(* IEC 61131-3 sources: elnaProjects/ElpcLogic/PomarKc7Changed/build_USO_ecl/_ (part 7) *)

  (* [A2-15, AI1-3]  TOpornoYpornogoPodshipnikaEDT_2 *)
  stAI_Ini(data_Ini := TRUE,  dLL := 0.0, dHL := 100.0,
  ISVALIDREF_HA := TRUE, ISVALIDREF_HW := TRUE, dHA := 80.0, dHW := 75.0, aperturFilter:= 0.5, dMaxChangeSpeed := 10.0,
  strAI := ai.Toy_podshipnika_EDT_2);
  inits := inits + BOOL_TO_UINT(stAI_Ini.Init);

  (********************************************* Модуль A3-1 ******************************************************)

  (* [A3-1, AI2-0]  TOpornoYpornogoPodshipnikaKolesaRedEDT_3 *)
  stAI_Ini(data_Ini := TRUE,  dLL := 0.0, dHL := 100.0,
  ISVALIDREF_HA := TRUE, ISVALIDREF_HW := TRUE, dHA := 80.0, dHW := 75.0, aperturFilter:= 0.5, dMaxChangeSpeed := 10.0,
  strAI := ai.Toy_podshipnika_kol_EDT_3);
  inits := inits + BOOL_TO_UINT(stAI_Ini.Init);

  (* [A3-1, AI2-1] TOpornoYpornogoPodshipnikaKolesaRedHT_4 *)
  stAI_Ini(data_Ini := TRUE,  dLL := 0.0, dHL := 100.0,
  ISVALIDREF_HA := TRUE, ISVALIDREF_HW := TRUE, dHA := 80.0, dHW := 75.0, aperturFilter:= 0.5, dMaxChangeSpeed := 10.0,
  strAI := ai.Toy_podshipnika_kol_EDT_4);
  inits := inits + BOOL_TO_UINT(stAI_Ini.Init);

  (* [A3-1, AI2-2] TOpornogoPodshipnikaShesterniReduktoraT_5 *)
  stAI_Ini(data_Ini := TRUE,  dLL := 0.0, dHL := 100.0,
  ISVALIDREF_HA := TRUE, ISVALIDREF_HW := TRUE, dHA := 80.0, dHW := 75.0, aperturFilter:= 0.5, dMaxChangeSpeed := 10.0,
  strAI := ai.Toy_podshipnika_shest_red_EDT_5);
  inits := inits + BOOL_TO_UINT(stAI_Ini.Init);

  (* [A3-1, AI2-3] TOpornogoPodshipnikaReduktoraHT_6 *)
  stAI_Ini(data_Ini := TRUE,  dLL := 0.0, dHL := 100.0,
  ISVALIDREF_HA := TRUE, ISVALIDREF_HW := TRUE, dHA := 80.0, dHW := 75.0, aperturFilter:= 0.5, dMaxChangeSpeed := 10.0,
  strAI := ai.Ty_podshipnika_red_EDT_6);
  inits := inits + BOOL_TO_UINT(stAI_Ini.Init);

  (********************************************* Модуль A3-2 ******************************************************)

  (* [A3-2, AI3-01]  TOpornoYpornogoPodshipnikaNagnetateljaT_7_1 *)
  stAI_Ini(data_Ini := TRUE,  dLL := 0.0, dHL := 100.0,
  ISVALIDREF_HA := TRUE, ISVALIDREF_HW := TRUE, dHA := 80.0, dHW := 75.0, aperturFilter:= 0.5, dMaxChangeSpeed := 10.0,
  strAI := ai.Ty_podshipnika_nagnet_EDT_7_1);
  inits := inits + BOOL_TO_UINT(stAI_Ini.Init);

  (* [A3-2, AI3-01]  TOpornoYpornogoPodshipnikaNagnetateljaT_7_2 *)
  stAI_Ini(data_Ini := TRUE,  dLL := 0.0, dHL := 100.0,
  ISVALIDREF_HA := TRUE, ISVALIDREF_HW := TRUE, dHA := 80.0, dHW := 75.0, aperturFilter:= 0.5, dMaxChangeSpeed := 10.0,
  strAI := ai.Ty_podshipnika_nagnet_EDT_7_2);
  inits := inits + BOOL_TO_UINT(stAI_Ini.Init);

  (* [A3-2, AI3-2]  TOpornoYpornogoPodshipnikaSvobodnogoKoncaNT_8_1 *)
  stAI_Ini(data_Ini := TRUE,  dLL := 0.0, dHL := 100.0,
  ISVALIDREF_HA := TRUE, ISVALIDREF_HW := TRUE, dHA := 80.0, dHW := 75.0, aperturFilter:= 0.5, dMaxChangeSpeed := 10.0,
  strAI := ai.Toy_podshipnika_svobod_konca_EDT_8_1);
  inits := inits + BOOL_TO_UINT(stAI_Ini.Init);

  (* [A3-2, AI3-2]  TOpornoYpornogoPodshipnikaSvobodnogoKoncaNT_8_2 *)
  stAI_Ini(data_Ini := TRUE,  dLL := 0.0, dHL := 100.0,
  ISVALIDREF_HA := TRUE, ISVALIDREF_HW := TRUE, dHA := 80.0, dHW := 75.0, aperturFilter:= 0.5, dMaxChangeSpeed := 10.0,
  strAI := ai.Toy_podshipnika_svobod_konca_EDT_8_2);
  inits := inits + BOOL_TO_UINT(stAI_Ini.Init);

  (********************************************* Модуль A3-3 ******************************************************)

  (* [A3-3, AI4-1]  TYpornogoPodshipnikaRavKolodokHT_9_1 *)
  stAI_Ini(data_Ini := TRUE,  dLL := 0.0, dHL := 100.0,
  ISVALIDREF_HA := TRUE, ISVALIDREF_HW := TRUE, dHA := 80.0, dHW := 75.0, aperturFilter:= 0.5, dMaxChangeSpeed := 10.0,
  strAI := ai.Toy_podshipnika_rab_kol_EDT_9_1);
  inits := inits + BOOL_TO_UINT(stAI_Ini.Init);

  (* [A3-3, AI4-1]  TYpornogoPodshipnikaRavKolodokHT_9_2 *)
  stAI_Ini(data_Ini := TRUE,  dLL := 0.0, dHL := 100.0,
  ISVALIDREF_HA := TRUE, ISVALIDREF_HW := TRUE, dHA := 80.0, dHW := 75.0, aperturFilter:= 0.5, dMaxChangeSpeed := 10.0,
  strAI := ai.Toy_podshipnika_rab_kol_EDT_9_2);
  inits := inits + BOOL_TO_UINT(stAI_Ini.Init);

  (* [A3-3, AI4-3] TYpornogoPodshipnikaNerabKolodokHT_10_1 *)
  stAI_Ini(data_Ini := TRUE,  dLL := 0.0, dHL := 100.0,
  ISVALIDREF_HA := TRUE, ISVALIDREF_HW := TRUE, dHA := 80.0, dHW := 75.0, aperturFilter:= 0.5, dMaxChangeSpeed := 10.0,
  strAI := ai.Toy_podshipnika_nerab_kol_EDT_10_1);
  inits := inits + BOOL_TO_UINT(stAI_Ini.Init);

  (* [A3-3, AI4-3] TYpornogoPodshipnikaNerabKolodokHT_10_2 *)
  stAI_Ini(data_Ini := TRUE,  dLL := 0.0, dHL := 100.0,
  ISVALIDREF_HA := TRUE, ISVALIDREF_HW := TRUE, dHA := 80.0, dHW := 75.0, aperturFilter:= 0.5, dMaxChangeSpeed := 10.0,
  strAI := ai.Toy_podshipnika_nerab_kol_EDT_10_2);
  inits := inits + BOOL_TO_UINT(stAI_Ini.Init);

  (********************************************* Модуль A3-4 ******************************************************)
  (* [A3-4, AI5-0] THolodnogoVozduhaEDKanall *)
  stAI_Ini(data_Ini := TRUE,  dLL := 0.0, dHL := 100.0,
  ISVALIDREF_HW := TRUE, dHW := 60.0, aperturFilter:= 0.5,
  strAI := ai.Tholodnogo_vozduha_ED_kanal_1);
  inits := inits + BOOL_TO_UINT(stAI_Ini.Init);

  (* [A3-4, AI5-1] THolodnogoVozduhaEDKanal2 *)
  stAI_Ini(data_Ini := TRUE,  dLL := 0.0, dHL := 100.0,
  ISVALIDREF_HW := TRUE, dHW := 60.0, aperturFilter:= 0.5,
  strAI := ai.Tholodnogo_vozduha_ED_kanal_2);
  inits := inits + BOOL_TO_UINT(stAI_Ini.Init);

  (* [A3-4, AI5-2]  TGorjachegoVozduhaEDKanall *)
  stAI_Ini(data_Ini := TRUE,  dLL := 0.0, dHL := 100.0,
  ISVALIDREF_HW := TRUE, dHW := 70.0, aperturFilter:= 0.5,
  strAI := ai.Tgorjachego_vozduha_ED_kanal_1);
  inits := inits + BOOL_TO_UINT(stAI_Ini.Init);

  (* [A3-4, AI5-3] TGorjachegoVozduhaEDKanal2 *)
  stAI_Ini(data_Ini := TRUE,  dLL := 0.0, dHL := 100.0,
  ISVALIDREF_HW := TRUE, dHW := 70.0, aperturFilter:= 0.5,
  strAI := ai.Tgorjachego_vozduha_ED_kanal_2);
  inits := inits + BOOL_TO_UINT(stAI_Ini.Init);

  (********************************************* Модуль A3-5 ******************************************************)

  (* [A3-5, AI6-0] TNArujnogoVozduha *)
  stAI_Ini(data_Ini := TRUE,  dLL := -50.0, dHL := 100.0,
  ISVALIDREF_HW := TRUE, dHW := 70.0, aperturFilter:= 0.5,
  strAI := ai.Tnarujnogo_vozduha);
  inits := inits + BOOL_TO_UINT(stAI_Ini.Init);

  (* [A3-5, AI6-1]  TgazaNaVhodeH *)
  stAI_Ini(data_Ini := TRUE,  dLL := -50.0, dHL := 100.0,
  ISVALIDREF_HW := TRUE, dHW := 80.0, aperturFilter:= 0.5,
  strAI := ai.Tgaza_na_vhode_H);
  inits := inits + BOOL_TO_UINT(stAI_Ini.Init);

  (* [A3-5, AI6-2] TgazaNaVyhodeH *)
  stAI_Ini(data_Ini := TRUE,  dLL := -50.0, dHL := 100.0,
  ISVALIDREF_HW := TRUE, ISVALIDREF_HA := TRUE, dHa :=90.0, dHW := 80.0, aperturFilter:= 0.5, dMaxChangeSpeed := 10.0,
  strAI := ai.Tgaza_na_vyhode_H);
  inits := inits + BOOL_TO_UINT(stAI_Ini.Init);

  (********************************************* Модуль A3-6 ******************************************************)
  (* [A3-6, AI7-0] TMasladoAVOM *)
  stAI_Ini(data_Ini := TRUE,  dLL := 0.0, dHL := 150.0,
  ISVALIDREF_HW := TRUE, dHW := 55.0, aperturFilter:= 0.5,
  strAI := ai.Tmasla_do_AVOM);
  inits := inits + BOOL_TO_UINT(stAI_Ini.Init);

  (* [A3-6, AI7-1] TMaslaPosleAVOM *)
  stAI_Ini(data_Ini := TRUE,  dLL := 0.0, dHL := 150.0,
  ISVALIDREF_HW := TRUE, dHW := 55.0, aperturFilter:= 0.5, dMaxChangeSpeed := 10.0,
  strAI := ai.Tmasla_posle_AVOM);
  inits := inits + BOOL_TO_UINT(stAI_Ini.Init);
  (********************************************* Модуль A3-8 ******************************************************)
  (* [A3-8, AI9-0]  TMaslaMB *)
  stAI_Ini(data_Ini := TRUE,  dLL := 0.0, dHL := 150.0,
  ISVALIDREF_LW := TRUE, dLW := 25.0, aperturFilter:= 0.5, dMaxChangeSpeed := 10.0,
  strAI := ai.Tmasla_MB);
  inits := inits + BOOL_TO_UINT(stAI_Ini.Init);

  (* [A3-6, AI7-2] TMaslaMB_TEN *)
  stAI_Ini(data_Ini := TRUE,  dLL := 0.0, dHL := 100.0,
  ISVALIDREF_HW := TRUE, dHW := 50.0, aperturFilter:= 0.5, dMaxChangeSpeed := 10.0,
  strAI := ai.Tmasla_MB_TEN);
  inits := inits + BOOL_TO_UINT(stAI_Ini.Init);

  (* [A3-8, AI9-1]  TEmperatura_v_SHU *)
  stAI_Ini(data_Ini := TRUE,  dLL := -40.0, dHL := 100.0, CurrentShotCircuit := 20320.0, CurrentBreakCircuit := 3680.0,
  aperturFilter:= 0.5, strAI := ai.Tshu);
  inits := inits + BOOL_TO_UINT(stAI_Ini.Init);

  (* [A3-8, AI9-2]  DavlenijaMasloSmNizkoe *)
  stAI_Ini(data_Ini := TRUE,  dLL := 0.0, dHL := 250.0,
  ISVALIDREF_LW := TRUE, ISVALIDREF_LA := TRUE, dLW := 50.0, dLA := 25.0,  CurrentShotCircuit := 20240.0, CurrentBreakCircuit := 3760.0,  aperturFilter:= 0.5,
  strAI := ai.Pmaslo_sm_nizkoe);
  inits := inits + BOOL_TO_UINT(stAI_Ini.Init);

  (* [A3-8, AI9-3]  PerepadDavlenieNaMasloFiltre *)
  stAI_Ini(data_Ini := TRUE,  dLL := 0.0, dHL := 250.0,
  ISVALIDREF_HW := TRUE, dHW := 150.0, CurrentShotCircuit := 20240.0, CurrentBreakCircuit := 3760.0, aperturFilter:= 0.5,
  strAI := ai.dPgaza_na_maslo_filtre);
  inits := inits + BOOL_TO_UINT(stAI_Ini.Init);

  (********************************************* Модуль A3-9 ******************************************************)
  (* [A3-9, AI10-0]  DavlenijaMasloSmVysokoe *)
  stAI_Ini(data_Ini := TRUE,  dLL := 0.0, dHL := 1000.0,
  ISVALIDREF_LW := TRUE, ISVALIDREF_LA := TRUE, dLW := 300.0, dLA := 250.0, CurrentShotCircuit := 20240.0, CurrentBreakCircuit := 3760.0, aperturFilter:= 0.5,
  strAI := ai.Pmaslo_sm_vysokoe);
  inits := inits + BOOL_TO_UINT(stAI_Ini.Init);

  (* [A3-9, AI10-1]  DavlenijaMaslaPosleGNS *)
  stAI_Ini(data_Ini := TRUE,  dLL := 0.0, dHL := 250.0, aperturFilter:= 0.5, CurrentShotCircuit := 20240.0, CurrentBreakCircuit := 3760.0,
  ISVALIDREF_LW := TRUE, ISVALIDREF_HW := TRUE,
  dLW := 187.0, dHW := 242.0,
  strAI := ai.Pmasla_posle_GNS);
  inits := inits + BOOL_TO_UINT(stAI_Ini.Init);

  (* [A3-9, AI10-2] DavlenijaMaslaPosleNU *)
  stAI_Ini(data_Ini := TRUE,  dLL := 0.0, dHL := 10.0, aperturFilter:= 0.5, CurrentShotCircuit := 20240.0, CurrentBreakCircuit := 3760.0,
  ISVALIDREF_LW := TRUE, dLW := 3.0,
  strAI := ai.Pmasla_posle_NU);
  inits := inits + BOOL_TO_UINT(stAI_Ini.Init);

  (********************************************* Модуль A3-10 ******************************************************)
  (* [A3-10, AI11-0] PerepadDavlenieNaKonfuzore *)
  stAI_Ini(data_Ini := TRUE,  dLL := 0.0, dHL := 250.0,
  ISVALIDREF_LW := TRUE, dLW := 15.0, aperturFilter:= 0.5, CurrentShotCircuit := 20240.0, CurrentBreakCircuit := 3760.0,
  strAI := ai.dPgaza_na_konfuzore);
  inits := inits + BOOL_TO_UINT(stAI_Ini.Init);

  (* [A3-10, AI11-1] OsSdvigNagnetatelja_Plus *)
  stAI_Ini(data_Ini := TRUE,  dLL := 0.0, dHL := 1000.0,
  ISVALIDREF_HA := TRUE, ISVALIDREF_HW := TRUE, dHW := 200.0, dHA := 300.0, aperturFilter := 0.5, CurrentShotCircuit := 20240.0, CurrentBreakCircuit := 3760.0,
  strAI := ai.Os_sdvig_nagnetatelja_plus);
  inits := inits + BOOL_TO_UINT(stAI_Ini.Init);

  (* [A3-10, AI11-2] OsSdvigNagnetatelja_Minus *)
  stAI_Ini(data_Ini := TRUE,  dLL := 0.0, dHL := 1600.0,
  ISVALIDREF_LW := TRUE, dLW := 150.0, ISVALIDREF_LA := TRUE, dLA := 100.0, aperturFilter := 0.5, CurrentShotCircuit := 20240.0, CurrentBreakCircuit := 3760.0,
  strAI := ai.Os_sdvig_nagnetatelja_minus);
  inits := inits + BOOL_TO_UINT(stAI_Ini.Init);

  (* [A3-10, AI11-3] PerepadDavlenieMasloGaz *)
  stAI_Ini(data_Ini := TRUE, dLL := 0.0, dHL := 1600.0,
  ISVALIDREF_LW := TRUE, ISVALIDREF_LA := TRUE, dLW := 150.0, dLa := 100.0, aperturFilter:= 0.5, CurrentShotCircuit := 20240.0, CurrentBreakCircuit := 3760.0,
  strAI := ai.dPmaslo_gaz);
  inits := inits + BOOL_TO_UINT(stAI_Ini.Init);

  (********************************************* Модуль A3-11 ******************************************************)
  (* [A3-11, AI12-0]  DGazaNaVhodeNagnetatelja *)
  stAI_Ini(data_Ini := TRUE,  dLL := 0.0, dHL := 10.0,
  ISVALIDREF_LW := TRUE, dLW := 4.895, aperturFilter := 0.5, CurrentShotCircuit := 20240.0, CurrentBreakCircuit := 3760.0,
  strAI := ai.Pgaza_na_vhode_nagnetatelia);
  inits := inits + BOOL_TO_UINT(stAI_Ini.Init);

  (* [A3-11, AI12-1]  DGazaNaVyhodeNagnetatelja *)
  stAI_Ini(data_Ini := TRUE,  dLL := 0.0, dHL := 10.0,
  ISVALIDREF_HA := TRUE, ISVALIDREF_HW := TRUE, dLA := 7.653, dHW := 7.55, aperturFilter := 0.5, CurrentShotCircuit := 20240.0, CurrentBreakCircuit := 3760.0,
  strAI := ai.Pgaza_na_vyhode_nagnetatelia);
  inits := inits + BOOL_TO_UINT(stAI_Ini.Init);

  (* [A3-11, AI12-3]  DavlenieImpulsGaz *)
  stAI_Ini(data_Ini := TRUE,  dLL := 0.0, dHL := 10.0,
  ISVALIDREF_LW := TRUE, dLW := 5.0, aperturFilter := 0.5, CurrentShotCircuit := 20240.0, CurrentBreakCircuit := 3760.0,
  strAI := ai.Pimpuls_gaz);
  inits := inits + BOOL_TO_UINT(stAI_Ini.Init);

  (********************************************* Модуль A3-12 ******************************************************)
  (* [A3-12, AI13-0] YrovenMaslaMB *)
  stAI_Ini(data_Ini := TRUE,  dLL := 190.0, dHL := 885.0,
  ISVALIDREF_LW := TRUE, dLW := 530.0, aperturFilter := 0.5,  CurrentShotCircuit := 20240.0, CurrentBreakCircuit := 3760.0,
  strAI := ai.Yroven_masla_MB);
  inits := inits + BOOL_TO_UINT(stAI_Ini.Init);

  (********************************************* Модуль A3-13 ******************************************************)
  (* [A3-13, AI14-0]  Kontrol_per220V *)
  stAI_Ini(data_Ini := TRUE,  dLL := 0.0, dHL := 250.0,
  ISVALIDREF_LW := TRUE, ISVALIDREF_HW := TRUE, dLW := 187.0, dHW := 242.0, aperturFilter := 0.5, CurrentShotCircuit := 20240.0, CurrentBreakCircuit := 3760.0,
  strAI := ai.Kontrol_per_220V);
  inits := inits + BOOL_TO_UINT(stAI_Ini.Init);

  (* [A3-13, AI14-1]  Kontrol_post220V *)
  stAI_Ini(data_Ini := TRUE,  dLL := 0.0, dHL := 250.0,
  ISVALIDREF_HW := TRUE, ISVALIDREF_LW := TRUE, dHW := 242.0, dLW := 187.0, aperturFilter := 0.5, CurrentShotCircuit := 20240.0, CurrentBreakCircuit := 3760.0,
  strAI := ai.Kontrol_post_220V);
  inits := inits + BOOL_TO_UINT(stAI_Ini.Init);

  (* [A3-13, AI14-2]  VibroSkorostOPED_T1 *)
  stAI_Ini(data_Ini := TRUE,  dLL := 0.0, dHL := 25.0,
  ISVALIDREF_HW := TRUE, ISVALIDREF_HA := TRUE, dHW := 11.0, dHA := 18.0, aperturFilter := 0.5, CurrentShotCircuit := 20240.0, CurrentBreakCircuit := 3760.0,
  strAI := ai.Vibro_skorost_OPED_T1);
  inits := inits + BOOL_TO_UINT(stAI_Ini.Init);

  (* [A3-13, AI14-3]  VibroSkorostOYPED_T2 *)
  stAI_Ini(data_Ini := TRUE,  dLL := 0.0, dHL := 25.0,
  ISVALIDREF_HW := TRUE, ISVALIDREF_HA := TRUE, dHW := 11.0, dHA := 18.0, aperturFilter := 0.5, CurrentShotCircuit := 20240.0, CurrentBreakCircuit := 3760.0,
  strAI := ai.Vibro_skorost_OYPED_T2);
  inits := inits + BOOL_TO_UINT(stAI_Ini.Init);

  (********************************************* Модуль A3-14 ******************************************************)
  (* [A3-14, AI15-0]  VibroSkorostOYPKolesaED_T3 *)
  stAI_Ini(data_Ini := TRUE,  dLL := 0.0, dHL := 25.0,
  ISVALIDREF_HW := TRUE, ISVALIDREF_HA := TRUE, dHW := 11.0, dHA := 18.0, aperturFilter := 0.5, CurrentShotCircuit := 20240.0, CurrentBreakCircuit := 3760.0,
  strAI := ai.Vibro_skorost_OYP_kolesa_ED_T3);
  inits := inits + BOOL_TO_UINT(stAI_Ini.Init);

  (* [A3-14, AI15-1]  VibroSkorostOPKolesaRH_T4 *)
  stAI_Ini(data_Ini := TRUE,  dLL := 0.0, dHL := 25.0,
  ISVALIDREF_HW := TRUE, ISVALIDREF_HA := TRUE, dHW := 11.0, dHA := 18.0, aperturFilter := 0.5, CurrentShotCircuit := 20240.0, CurrentBreakCircuit := 3760.0,
  strAI := ai.Vibro_skorost_OP_kolesa_RH_T4);
  inits := inits + BOOL_TO_UINT(stAI_Ini.Init);

  (* [A3-11, AI12-2]  VibroSkorostOPShesterniRED_T5 *)
  stAI_Ini(data_Ini := TRUE,  dLL := 0.0, dHL := 25.0,
  ISVALIDREF_HW := TRUE, ISVALIDREF_HA := TRUE, dHW := 11.0, dHA := 18.0, aperturFilter := 0.5, CurrentShotCircuit := 20240.0, CurrentBreakCircuit := 3760.0,
  strAI := ai.Vibro_skorost_OP_shesterni_RED_T5);
  inits := inits + BOOL_TO_UINT(stAI_Ini.Init);

  (* [A3-11, AI12-2]  VibroSkorostOPShesterniRED_T5 *)
  stAI_Ini(data_Ini := TRUE,  dLL := 0.0, dHL := 25.0,
  ISVALIDREF_HW := TRUE, ISVALIDREF_HA := TRUE, dHW := 11.0, dHA := 18.0, aperturFilter := 0.5, CurrentShotCircuit := 20240.0, CurrentBreakCircuit := 3760.0,
  strAI := ai.Vibro_skorost_OP_shesterni_RED_T6);
  inits := inits + BOOL_TO_UINT(stAI_Ini.Init);

  (* [A3-11, AI12-2]  VibroSkorostOPShesterniRED_T5 *)
  stAI_Ini(data_Ini := TRUE,  dLL := 0.0, dHL := 1000.0,
  ISVALIDREF_LW := TRUE, dLW := 300.0, aperturFilter := 0.5, CurrentShotCircuit := 20240.0, CurrentBreakCircuit := 3760.0,
  strAI := ai.Tok_statora);
  inits := inits + BOOL_TO_UINT(stAI_Ini.Init);

  initiales := 0;
  IF init THEN initiales := inits; END_IF;
END_FUNCTION_BLOCK

FUNCTION_BLOCK fb_AiSourceMlp_timer
  VAR_INPUT
    arAIN : TItemAIN;
    err_mod : TItemDIN;
  END_VAR
  VAR_IN_OUT
    strAI : struct_AI;
  END_VAR
  VAR
    _statusAi : TYPE_StatusAi;
    _commandAnalog : TYPE_CommandAnalog;
    _sunpackerCommand : fb_sunpackerCommand;
    _AnalogLimitFlags : TYPE_AnalogLimitFlags;
    notReliable : BOOL;
    _lastValue : LREAL;
    resetCmdTimer : TON;
    _LastValueTimer : TON;
    resetCmdTimerPriznak : BOOL;
    k : LREAL;
    b : LREAL;
    ap : LREAL;
    raznitsa : LREAL;
    rABS : LREAL;
    h : LREAL;
    mismatch : LREAL;
    parametr : BYTE;
    source : BYTE;
    cmd : BYTE;
    lastCmd : BYTE;
    source_for_Status : BYTE;
    cmd_for_Status : BYTE;
    command_error_for_Status : BYTE;
    secondTakt : BOOL;
    off_trig : R_TRIG;
    on_trig : R_TRIG;
    remont_trig : R_TRIG;
    LL_trig : R_TRIG;
    HL_trig : R_TRIG;
    Normal_trig : R_TRIG;
    Nedostover_trig : R_TRIG;
    timerLA : TON;
    timerHA : TON;
    timerLW : TON;
    timerHW : TON;
  END_VAR
  VAR RETAIN
    retainLL : LREAL;
    retainHL : LREAL;
    retainLA : LREAL;
    retainHA : LREAL;
    retainLW : LREAL;
    retainHW : LREAL;
  END_VAR

  strAI.opcCommandsDisabled := strAI.inopcCommandsDisabled ;

  (* ---- При первом пуске принимаем значение уставок ---- *)
  IF NOT secondTakt THEN
            IF (strAI.dLL <> retainLL) AND (retainLL <> 0.0) THEN  strAI.LL := retainLL;
            ELSE strAI.LL := strAI.dLL; END_IF;
  	IF (strAI.dHL <> retainHL) AND (retainHL <> 0.0) THEN  strAI.HL := retainHL;
            ELSE strAI.HL := strAI.dHL; END_IF;

            IF strAI.ISVALIDREF_HA AND (strAI.dHA <> retainHA) AND (retainHA <> 0.0) THEN  strAI.HA := retainHA;
            ELSE strAI.HA := strAI.dHA; END_IF;

            IF strAI.ISVALIDREF_LA AND (strAI.dLA <> retainLA) AND (retainLA <> 0.0) THEN  strAI.LA := retainLA;
            ELSE strAI.LA := strAI.dLA; END_IF;

            IF strAI.ISVALIDREF_HW AND (strAI.dHW <> retainHW) AND (retainHW <> 0.0) THEN  strAI.HW := retainHW;
            ELSE strAI.HW := strAI.dHW; END_IF;

            IF strAI.ISVALIDREF_LW AND (strAI.dLW <> retainLW) AND (retainLW <> 0.0) THEN  strAI.LW := retainLW;
            ELSE strAI.LW := strAI.dLW; END_IF;

  	secondTakt  := TRUE;
  END_IF;

  (* ---- пересчет тока в физ величину ---- *)
  k := (strAI.HL - strAI.LL)/(strAI.inpHl - strAI.inpLL);
  b := strAI.LL - k * strAI.inpLL;
  strAI.value := k * arAIN.dblValue + b;

  (* ---- определение обрыва и кз ----- *)

  strAI.blConnect := true;(*(UINT_TO_WORD(arAIN.wFlags) = 1472) and (UINT_TO_WORD(err_mod.wValue) = 20) and (UINT_TO_WORD(err_mod.wFlags) = 192); *)
  IF NOT strAI.blConnect THEN
      strAI.interval := _statusAi.NOTDEFINED;
  ELSIF ((arAIN.dblValue < strAI.currentBreakCircuit) AND (strAI.currentBreakCircuit > 0.0)) OR ((strAI.interval = _statusAi.LL) AND (arAIN.dblValue < (strAI.currentBreakCircuit + 100.0))) THEN
      strAI.interval := _statusAi.LL;
  ELSIF ((arAIN.dblValue > strAI.currentShotCircuit) AND (strAI.currentShotCircuit > 0.0)) OR ((strAI.interval = _statusAi.HL) AND (arAIN.dblValue > (strAI.currentShotCircuit - 100.0))) THEN
      strAI.interval := _statusAi.HL;
  ELSE
      strAI.interval := _statusAi.normal;
  END_IF;

  IF NOT strAI.imit THEN
  	(* Расчет апертурного фильтра*)
  	ap := strAI.aperturFilter * 0.01 * (strAI.HL - strAI.LL);
  	IF strAI.aperturFilter <> 0.0 THEN raznitsa := strAI.value- _lastValue;
  		IF 	raznitsa < 0.0 	THEN 	rABS := -raznitsa; 		ELSE 	rABS := raznitsa; 		END_IF;
  		IF 	rABS > ap 	THEN 	strAI.value := strAI.value;	ELSE 	strAI.value := _lastValue; 	END_IF;
  	END_IF;

  	(* Расчет экпоненциального фильтра*)
  	IF strAI.exponentialFilter <> 0.0 THEN strAI.value := (strAI.exponentialFilter * strAI.value) + ((1.0 - strAI.exponentialFilter) * _lastValue); END_IF;
  ELSE
  	strAI.interval := _statusAi.normal;
  END_IF;

  IF notReliable THEN strAI.interval := _statusAi.NOTRELIABLE; END_IF;

  IF NOT notReliable THEN
  	IF strAI.interval >= _statusAi.normal THEN
  		strAI.interval := _statusAi.NOTDEFINED;
  		h := strAI.histeresis* 0.01 * (strAI.HL-strAI.LL);
  		(*определение выхода за аппаратные границы вынесено в GetData.здесь только для нужд имитации*)
  		IF strAI.imit THEN
  			mismatch := strAI.rassoglasovanie * 0.01 * (strAI.HL - strAI.LL);
  			IF ( strAI.value < strAI.LL - mismatch)   THEN strAI.interval := _statusAi.LL;
  			ELSIF  (strAI.value > strAI.Hl + mismatch) THEN strAI.interval := _statusAi.HL; END_IF;
  		ELSE
  			strAI.interval := _statusAi.normal;
  			IF strAI.ISVALIDREF_LA AND NOT strAI.Disabled_LA AND (strAI.interval = _statusAi.normal) THEN
                                timerLA(IN:=(strAI.value  < strAI.LA) OR ((strAI.interval = _statusAi.LA)  AND ((strAI.value - h) < strAI.LA)), PT:=strAI.delayLA);
  				IF timerLA.Q  THEN
  					strAI.interval := _statusAi.LA;
  				END_IF;
  			END_IF;
  			IF strAI.ISVALIDREF_HA  AND NOT strAI.Disabled_HA AND (strAI.interval = _statusAi.normal)  THEN
                                timerHA(IN:=(strAI.value > strAI.HA) OR ((strAI.interval = _statusAi.HA)  AND ((strAI.value + h) > strAI.HA)), PT:=strAI.delayHA);
  				IF timerHA.Q  THEN
  					strAI.interval := _statusAi.HA;
  				END_IF;
  			END_IF;
  			IF strAI.ISVALIDREF_LW AND NOT strAI.Disabled_LW AND (strAI.interval = _statusAi.normal)  THEN
                                timerLW(IN:=(strAI.value < strAI.LW) OR ((strAI.interval = _statusAi.LW)  AND ((strAI.value - h) < strAI.LW)), PT:=strAI.delayLW);
  				IF timerLW.Q THEN
  					strAI.interval := _statusAi.LW;
  				END_IF;
  			END_IF;
  			IF strAI.ISVALIDREF_HW AND NOT strAI.Disabled_HW  AND (strAI.interval = _statusAi.normal) THEN
                                timerHW(IN:=(strAI.value > strAI.HW)  OR ((strAI.interval = _statusAi.HW)  AND ((strAI.value + h) > strAI.HW)), PT:=strAI.delayHW);
  				IF  timerHW.Q  THEN
  					strAI.interval := _statusAi.HW;
  				END_IF;
  			END_IF;
  		END_IF;
  	END_IF;
  ELSE
  	strAI.interval := _statusAi.NOTRELIABLE;
  END_IF;

  IF strAI.remont THEN strAI.interval := _statusAi.NOTDEFINED; END_IF;

  _sunpackerCommand(command := strAI.inCommand);
  	source := _sunpackerCommand.source;
  	parametr := _sunpackerCommand.parametr;
  	cmd := _sunpackerCommand.cmd;

  IF cmd <> 0 AND lastCmd <> cmd and (((NOT strAI.opcCommandsDisabled) AND source > 0) OR source = 0) then
  	CASE BYTE_TO_INT(cmd) OF
  	(*cmd_SetUstavki*) 1 :
  				IF ((parametr AND _AnalogLimitFlags.LL) <> 0)		             	THEN 	strAI.LL := strAI.dLL; retainLL:= strAI.LL; END_IF;
  				IF ((parametr AND _AnalogLimitFlags.HL) <> 0)		 	          THEN	strAI.HL := strAI.dHL; retainHL:= strAI.HL; END_IF;
  				IF ((parametr AND _AnalogLimitFlags.LA) <> 0) AND strAI.ISVALIDREF_LA 	THEN	strAI.LA := strAI.dLA; retainLA:= strAI.LA; END_IF;
  				IF ((parametr AND _AnalogLimitFlags.HA) <> 0) AND strAI.ISVALIDREF_HA 	THEN	strAI.HA := strAI.dHA; retainHA:= strAI.HA; END_IF;
  				IF ((parametr AND _AnalogLimitFlags.LW) <> 0) AND strAI.ISVALIDREF_LW 	THEN	strAI.LW := strAI.dLW; retainLW:= strAI.LW; END_IF;
  				IF ((parametr AND _AnalogLimitFlags.HW) <> 0) AND strAI.ISVALIDREF_HW 	THEN	strAI.HW := strAI.dHW; retainHW:= strAI.HW; END_IF;
  	(*cmd_SetRemont*) 2 :
  				strAI.remont := TRUE;
  	(*cmd_ResetRemont*) 3 :
  				strAI.remont := FALSE;
  	(*cmd_kvitNotReliable*) 4 :
  				notReliable := FALSE;
  	END_CASE;
  	source_for_Status := source;
  	cmd_for_Status := cmd;
  	command_error_for_Status := 0;
  	resetCmdTimer(IN := FALSE);
  	resetCmdTimerPriznak := TRUE;
  END_IF;
  lastCmd := cmd;

  resetCmdTimer(IN := resetCmdTimerPriznak, PT := T#5S);
  IF resetCmdTimer.Q THEN
  	resetCmdTimerPriznak := FALSE;
  	source_for_Status := 0;
  	cmd_for_Status := 0;
  	command_error_for_Status := 0;
  END_IF;

  strAI.NS_Min := (strAI.value < strAI.minValue) AND strAI.minValue_ISVALIDREF;
  strAI.NS_Max := (strAI.value > strAI.maxValue) AND strAI.maxValue_ISVALIDREF;

  strAI.NS := (strAI.interval <= _statusAi.normal) AND NOT strAI.remont;

  Normal_trig(CLK := strAI.interval >= _statusAi.normal);

  IF NOT Normal_trig.Q THEN
  	_LastValueTimer(PT := T#1S);
  	IF (strAI.value<>_lastValue) OR _LastValueTimer.Q THEN
  		IF (_LastValueTimer.ET>T#0MS) THEN
  			strAI.ChangeSpeed:=(strAI.value-_lastValue)/(TIME_TO_LREAL(_LastValueTimer.ET)/1000.0);
  		END_IF;
  		_LastValueTimer(IN:=FALSE);

  		_LastValueTimer(IN:=TRUE);
  	END_IF;
  END_IF;
  _lastValue := strAI.value;

  IF ((strAI.maxChangeSpeed<>0.0) OR  (strAI.maxChangeSpeedDown<>0.0)) AND ( strAI.interval>=_statusAi.normal) THEN
  		IF (strAI.ChangeSpeed>0.0) THEN
  		    IF (strAI.ChangeSpeed > strAI.maxChangeSpeed) AND (strAI.maxChangeSpeed>0.0000001) THEN
  			 notReliable:=TRUE;
  		    END_IF;
  		ELSE
  		    IF (ABS(strAI.ChangeSpeed)>strAI.maxChangeSpeedDown) AND (strAI.maxChangeSpeedDown>0.0000001)  THEN
                                 notReliable:=TRUE;
  		    END_IF;
  		END_IF;

  END_IF;

  strAI.status := SHL(BYTE_TO_DWORD(source_for_Status), 29) 		              (* Источник команды *)
  			OR SHL(BYTE_TO_DWORD(cmd_for_Status), 26) 	    (* Команда *)
  			OR SHL(BYTE_TO_DWORD(command_error_for_Status), 23)   (* Ошибка команды *)
  			OR SHL(BOOL_TO_DWORD(strAI.OpcCommandsDisabled ), 21) (* Управление в ВУ заблокировано *)
  			OR SHL(BOOL_TO_DWORD(strAI.Disabled_HA), 9)		    (* ВА исключена из формирования интервала *)
  			OR SHL(BOOL_TO_DWORD(strAI.Disabled_LA), 8)		    (* НА исключена из формирования интервала *)
  			OR SHL(BOOL_TO_DWORD(strAI.Disabled_HW), 7)		    (* ВП исключена из формирования интервала *)
  			OR SHL(BOOL_TO_DWORD(strAI.Disabled_LW), 6)	              (* НП исключена из формирования интервала *)
  			OR SHL(BOOL_TO_DWORD(strAI.NS), 5)			    (* неиспарвность сигнала *)
  			OR SHL(BOOL_TO_DWORD(strAI.remont), 4)	              (* Выведен в ремонт *)
  			OR BYTE_TO_DWORD(strAI.interval);	              (* интервал *)
END_FUNCTION_BLOCK

FUNCTION_BLOCK proc_AI
  VAR
    fb_TStalisStatoraKanal1 : fb_AiSourceMlp;
    fb_TStalisStatoraKanal2 : fb_AiSourceMlp;
    fb_TStalisStatoraKanal3 : fb_AiSourceMlp;
    fb_TMediStatoraKanal1 : fb_AiSourceMlp;
    fb_TMediStatoraKanal2 : fb_AiSourceMlp;
    fb_TMediStatoraKanal3 : fb_AiSourceMlp;
    fb_TOpornogoPodshipnikaEDT_1 : fb_AiSourceMlp;
    fb_TOpornoYpornogoPodshipnikaEDT_2 : fb_AiSourceMlp;
    fb_TOpornoYpornogoPodshipnikaKolesaRedEDT_3 : fb_AiSourceMlp;
    fb_TOpornoYpornogoPodshipnikaKolesaRedHT_4 : fb_AiSourceMlp;
    fb_TOpornogoPodshipnikaShesterniReduktoraT_5 : fb_AiSourceMlp;
    fb_TOpornogoPodshipnikaReduktoraHT_6 : fb_AiSourceMlp;
    fb_TOpornoYpornogoPodshipnikaNagnetateljaT_7_1 : fb_AiSourceMlp;
    fb_TOpornoYpornogoPodshipnikaNagnetateljaT_7_2 : fb_AiSourceMlp;
    fb_TOpornoYpornogoPodshipnikaSvobodnogoKoncaNT_8_1 : fb_AiSourceMlp;
    fb_TOpornoYpornogoPodshipnikaSvobodnogoKoncaNT_8_2 : fb_AiSourceMlp;
    fb_TYpornogoPodshipnikaRabKolodokHT_9_1 : fb_AiSourceMlp;
    fb_TYpornogoPodshipnikaRabKolodokHT_9_2 : fb_AiSourceMlp;
    fb_TYpornogoPodshipnikYstanKolodokHT_10_1 : fb_AiSourceMlp;
    fb_TYpornogoPodshipnikYstanKolodokHT_10_2 : fb_AiSourceMlp;
    fb_THolodnogoVozduhaEDKanall : fb_AiSourceMlp;
    fb_THolodnogoVozduhaEDKanal2 : fb_AiSourceMlp;
    fb_TGorjachegoVozduhaEDKanall : fb_AiSourceMlp;
    fb_TGorjachegoVozduhaEDKanal2 : fb_AiSourceMlp;
    fb_TNArujnogoVozduha : fb_AiSourceMlp;
    fb_TgazaNaVhodeH : fb_AiSourceMlp_timer;
    fb_TgazaNaVyhodeH : fb_AiSourceMlp;
    fb_TMasladoAVOM : fb_AiSourceMlp;
    fb_TMaslaPosleAVOM : fb_AiSourceMlp;
    fb_TMaslaMB : fb_AiSourceMlp;
    fb_TEmperatura_v_SHU : fb_AiSourceMlp_timer;
    fb_DavlenijaMasloSmNizkoe : fb_AiSourceMlp;
    fb_PerepadDavlenieNaMasloFiltre : fb_AiSourceMlp;
    fb_DavlenijaMasloSmVysokoe : fb_AiSourceMlp;
    fb_DavlenijaMaslaPosleGNS : fb_AiSourceMlp;
    fb_DavlenijaMaslaPosleNU : fb_AiSourceMlp;
    fb_PerepadDavlenieNaKonfuzore : fb_AiSourceMlp;
    fb_OsSdvigNagnetatelja_Plus : fb_AiSourceMlp;
    fb_OsSdvigNagnetatelja_Minus : fb_AiSourceMlp;
    fb_PerepadDavlenieMasloGaz : fb_AiSourceMlp;
    fb_VibroSkorostOYPKolesaED_T3 : fb_AiSourceMlp;
    fb_DGazaNaVhodeNagnetatelja : fb_AiSourceMlp;
    fb_DGazaNaVyhodeNagnetatelja : fb_AiSourceMlp;
    fb_DavlenieImpulsGaz : fb_AiSourceMlp;
    fb_YrovenMaslaMB : fb_AiSourceMlp;
    fb_Kontrol_per220V : fb_AiSourceMlp;
    fb_Kontrol_post220V : fb_AiSourceMlp;
    fb_TMaslaMB_TEN : fb_AiSourceMlp;
    fb_VibroSkorostOPED_T1 : fb_AiSourceMlp;
    fb_VibroSkorostOYPED_T2 : fb_AiSourceMlp;
    fb_VibroSkorostOPKolesaRH_T4 : fb_AiSourceMlp;
    fb_VibroSkorostOPShesterniRED_T5 : fb_AiSourceMlp;
    fb_VibroSkorostOPShesterniReduktoraH_T6 : fb_AiSourceMlp;
    fb_TokStatora : fb_AiSourceMlp;
  END_VAR
  VAR_EXTERNAL
    arAIN_0 : TItemAIN;
    arAIN_1 : TItemAIN;
    arAIN_2 : TItemAIN;
    arAIN_3 : TItemAIN;
    arAIN_4 : TItemAIN;
    arAIN_5 : TItemAIN;
    arAIN_6 : TItemAIN;
    arAIN_7 : TItemAIN;
    arAIN_8 : TItemAIN;
    arAIN_9 : TItemAIN;
    arAIN_10 : TItemAIN;
    arAIN_11 : TItemAIN;
    arAIN_12 : TItemAIN;
    arAIN_13 : TItemAIN;
    arAIN_14 : TItemAIN;
    arAIN_15 : TItemAIN;
    ai : AiConfig;
    arAIN_16 : TItemAIN;
    arAIN_17 : TItemAIN;
    arAIN_18 : TItemAIN;
    arAIN_19 : TItemAIN;
    arAIN_20 : TItemAIN;
    arAIN_21 : TItemAIN;
    arAIN_22 : TItemAIN;
    arAIN_23 : TItemAIN;
    arAIN_24 : TItemAIN;
    arAIN_25 : TItemAIN;
    arAIN_26 : TItemAIN;
    arAIN_27 : TItemAIN;
    arAIN_28 : TItemAIN;
    arAIN_29 : TItemAIN;
    arAIN_30 : TItemAIN;
    arAIN_31 : TItemAIN;
    arAIN_32 : TItemAIN;
    arAIN_33 : TItemAIN;
    arAIN_34 : TItemAIN;
    arAIN_35 : TItemAIN;
    arAIN_36 : TItemAIN;
    arAIN_37 : TItemAIN;
    arAIN_38 : TItemAIN;
    arAIN_39 : TItemAIN;
    arAIN_40 : TItemAIN;
    arAIN_41 : TItemAIN;
    arAIN_42 : TItemAIN;
    arAIN_43 : TItemAIN;
    arAIN_44 : TItemAIN;
    arAIN_45 : TItemAIN;
    arAIN_46 : TItemAIN;
    arAIN_47 : TItemAIN;
    arAIN_48 : TItemAIN;
    arAIN_49 : TItemAIN;
    arAIN_50 : TItemAIN;
    arAIN_51 : TItemAIN;
    arAIN_52 : TItemAIN;
    arAIN_53 : TItemAIN;
    arAIN_54 : TItemAIN;
    arAIN_55 : TItemAIN;
    arAIN_56 : TItemAIN;
    arAIN_57 : TItemAIN;
    arAIN_58 : TItemAIN;
    arAIN_59 : TItemAIN;
    arAIN_60 : TItemAIN;
    arAIN_61 : TItemAIN;
    arAIN_62 : TItemAIN;
    arAIN_63 : TItemAIN;
    arAIN_64 : TItemAIN;
    arAIN_65 : TItemAIN;
    arERR_3 : TItemDIN;
    arERR_4 : TItemDIN;
    arERR_5 : TItemDIN;
    arERR_6 : TItemDIN;
    arERR_7 : TItemDIN;
    arERR_8 : TItemDIN;
    arERR_9 : TItemDIN;
    A1_10_err_mode : UINT;
    A1_11_err_mode : UINT;
    A1_4_err_mode : UINT;
    A1_5_err_mode : UINT;
    A1_6_err_mode : UINT;
    A1_7_err_mode : UINT;
    A1_8_err_mode : UINT;
    A1_9_err_mode : UINT;
    A2_2_err_mode : UINT;
    A2_3_err_mode : UINT;
    AI_0_dblValue : LREAL;
    AI_10_dblValue : LREAL;
    AI_11_dblValue : LREAL;
    AI_12_dblValue : LREAL;
    AI_13_dblValue : LREAL;
    AI_14_dblValue : LREAL;
    AI_15_dblValue : LREAL;
    AI_16_dblValue : LREAL;
    AI_17_dblValue : LREAL;
    AI_18_dblValue : LREAL;
    AI_19_dblValue : LREAL;
    AI_1_dblValue : LREAL;
    AI_20_dblValue : LREAL;
    AI_21_dblValue : LREAL;
    AI_22_dblValue : LREAL;
    AI_23_dblValue : LREAL;
    AI_24_dblValue : LREAL;
    AI_25_dblValue : LREAL;
    AI_26_dblValue : LREAL;
    AI_27_dblValue : LREAL;
    AI_28_dblValue : LREAL;
    AI_29_dblValue : LREAL;
    AI_2_dblValue : LREAL;
    AI_30_dblValue : LREAL;
    AI_31_dblValue : LREAL;
    AI_32_dblValue : LREAL;
    AI_33_dblValue : LREAL;
    AI_34_dblValue : LREAL;
    AI_35_dblValue : LREAL;
    AI_36_dblValue : LREAL;
    AI_37_dblValue : LREAL;
    AI_38_dblValue : LREAL;
    AI_39_dblValue : LREAL;
    AI_3_dblValue : LREAL;
    AI_40_dblValue : LREAL;
    AI_41_dblValue : LREAL;
    AI_42_dblValue : LREAL;
    AI_43_dblValue : LREAL;
    AI_44_dblValue : LREAL;
    AI_45_dblValue : LREAL;
    AI_46_dblValue : LREAL;
    AI_47_dblValue : LREAL;
    AI_48_dblValue : LREAL;
    AI_49_dblValue : LREAL;
    AI_4_dblValue : LREAL;
    AI_50_dblValue : LREAL;
    AI_51_dblValue : LREAL;
    AI_52_dblValue : LREAL;
    AI_53_dblValue : LREAL;
    AI_54_dblValue : LREAL;
    AI_55_dblValue : LREAL;
    AI_56_dblValue : LREAL;
    AI_57_dblValue : LREAL;
    AI_58_dblValue : LREAL;
    AI_59_dblValue : LREAL;
    AI_5_dblValue : LREAL;
    AI_60_dblValue : LREAL;
    AI_61_dblValue : LREAL;
    AI_62_dblValue : LREAL;
    AI_63_dblValue : LREAL;
    AI_64_dblValue : LREAL;
    AI_65_dblValue : LREAL;
    AI_66_dblValue : LREAL;
    AI_67_dblValue : LREAL;
    AI_68_dblValue : LREAL;
    AI_69_dblValue : LREAL;
    AI_6_dblValue : LREAL;
    AI_70_dblValue : LREAL;
    AI_71_dblValue : LREAL;
    AI_72_dblValue : LREAL;
    AI_73_dblValue : LREAL;
    AI_74_dblValue : LREAL;
    AI_75_dblValue : LREAL;
    AI_76_dblValue : LREAL;
    AI_77_dblValue : LREAL;
    AI_78_dblValue : LREAL;
    AI_79_dblValue : LREAL;
    AI_7_dblValue : LREAL;
    AI_8_dblValue : LREAL;
    AI_9_dblValue : LREAL;
  END_VAR

  (* Циклический опрос. Входные аналоговые параметры *)

  (* [A1-9, AI5-4]  dР газа на конфузоре *)
  fb_PerepadDavlenieNaKonfuzore(arAIN := arAIN_40, strAI := ai.dPgaza_na_konfuzore, err_mod:=arERR_8);
  AI_40_dblValue := arAIN_40.dblValue;

  (* [A1-9, AI5-0] dР масла на масляном фильтре *)
  fb_PerepadDavlenieNaMasloFiltre(arAIN := arAIN_34, strAI := ai.dPgaza_na_maslo_filtre, err_mod:=arERR_8);
  AI_34_dblValue := arAIN_34.dblValue;

  (* [A1-9, AI5-7]  dР масло-газ *)
  fb_PerepadDavlenieMasloGaz(arAIN := arAIN_41, strAI := ai.dPmaslo_gaz, err_mod:=arERR_8);
  AI_41_dblValue := arAIN_41.dblValue;

  (* [A1-10, AI6-2] Р газа на входе нагнетателя *)
  fb_DGazaNaVhodeNagnetatelja(arAIN := arAIN_44, strAI := ai.Pgaza_na_vhode_nagnetatelia, err_mod:=arERR_9);
  AI_44_dblValue := arAIN_44.dblValue;

  (* [A1-10, AI6-3] Р газа на выходе нагнетателя *)
  fb_DGazaNaVyhodeNagnetatelja(arAIN := arAIN_45, strAI := ai.Pgaza_na_vyhode_nagnetatelia, err_mod:=arERR_9);
  AI_45_dblValue := arAIN_45.dblValue;

  (* [A1-9, AI5-3]  Р масла после НУ *)
  fb_DavlenijaMaslaPosleNU(arAIN := arAIN_37, strAI := ai.Pmasla_posle_NU, err_mod:=arERR_8);
  AI_37_dblValue := arAIN_37.dblValue;

  (* [A1-8, AI4-6]  Р масла смазки низкое) *)
  fb_DavlenijaMasloSmNizkoe(arAIN := arAIN_33, strAI := ai.Pmaslo_sm_nizkoe, err_mod:=arERR_7);
  AI_33_dblValue := arAIN_33.dblValue;

  (* [A1-9, AI5-2]  Р масла смазки после ГМНС *)
  fb_DavlenijaMaslaPosleGNS(arAIN := arAIN_36, strAI := ai.Pmasla_posle_GNS, err_mod:=arERR_8);
  AI_36_dblValue := arAIN_36.dblValue;

  (* [A1-9, AI5-1]  Р масла смазки высокое *)
  fb_DavlenijaMasloSmVysokoe(arAIN := arAIN_35, strAI := ai.Pmaslo_sm_vysokoe, err_mod:=arERR_8);
  AI_35_dblValue := arAIN_35.dblValue;

  (* [A1-7, AI3-2] Т наружного воздуха *)
  fb_TNArujnogoVozduha(arAIN := arAIN_24, strAI := ai.Tnarujnogo_vozduha, err_mod:=arERR_6);
  AI_24_dblValue := arAIN_24.dblValue;

  (* [A1-8, AI4-0]  Т газа на входе нагнетателя *)
  fb_TgazaNaVhodeH(arAIN := arAIN_25, strAI := ai.Tgaza_na_vhode_H, err_mod:=arERR_7);
  AI_25_dblValue := arAIN_25.dblValue;

  (* [A1-8, AI4-1] Т газа на выходе нагнетателя *)
  fb_TgazaNaVyhodeH(arAIN := arAIN_26, strAI := ai.Tgaza_na_vyhode_H, err_mod:=arERR_7);
  AI_26_dblValue := arAIN_26.dblValue;

  (* [A1-6, AI2-7]  Т горячего воздуха в ЭД, точка 1 *)
  fb_TGorjachegoVozduhaEDKanall(arAIN := arAIN_22, strAI := ai.Tgorjachego_vozduha_ED_kanal_1, err_mod:=arERR_5);
  AI_22_dblValue := arAIN_22.dblValue;

  (* [A1-7, AI3-0] Т горячего воздуха в ЭД, точка 2 *)
  fb_TGorjachegoVozduhaEDKanal2(arAIN := arAIN_23, strAI := ai.Tgorjachego_vozduha_ED_kanal_2, err_mod:=arERR_6);
  AI_23_dblValue := arAIN_23.dblValue;

  (* [A1-8, AI4-4] Т масла в маслобаке *)
  fb_TMaslaMB(arAIN := arAIN_29, strAI := ai.Tmasla_MB, err_mod:=arERR_7);
  AI_29_dblValue := arAIN_29.dblValue;

  (* [A1-8, AI4-4] Т масла в маслобаке над ТЭНом *)
  fb_TMaslaMB_TEN(arAIN := arAIN_30, strAI := ai.Tmasla_MB_TEN, err_mod:=arERR_7);
  AI_30_dblValue := arAIN_30.dblValue;

  (* [A1-8, AI4-2] Т масла до АВО М *)
  fb_TMasladoAVOM(arAIN := arAIN_27, strAI := ai.Tgorjachego_vozduha_ED_kanal_2, err_mod:=arERR_7);
  AI_27_dblValue := arAIN_27.dblValue;

  (* [A1-8, AI4-3] Т масла после АВО М *)
  fb_TMaslaPosleAVOM(arAIN := arAIN_28, strAI := ai.Tmasla_posle_AVOM, err_mod:=arERR_7);
  AI_28_dblValue := arAIN_28.dblValue;

  (* [A1-4, AI0-3] Т Т меди статора фаза 1 *)
  fb_TMediStatoraKanal1(arAIN := arAIN_3, strAI := ai.Tmedi_statora_kanal_1, err_mod:=arERR_3);
  AI_3_dblValue := arAIN_3.dblValue;

  (* [A1-4, AI0-4] Т обмотки фазы 3 канал *)
  fb_TMediStatoraKanal2(arAIN := arAIN_4, strAI := ai.Tmedi_statora_kanal_2, err_mod:=arERR_3);
  AI_4_dblValue := arAIN_4.dblValue;

  (* [A1-4, AI0-5] Т меди статора фаза 2 *)
  fb_TMediStatoraKanal3(arAIN := arAIN_5, strAI := ai.Tmedi_statora_kanal_3, err_mod:=arERR_3);
  AI_5_dblValue := arAIN_5.dblValue;

  (* [A1-4, AI0-6] Т ОП ЭД со стороны свободного конца (т.1) } *)
  fb_TOpornogoPodshipnikaEDT_1(arAIN := arAIN_6, strAI := ai.Toporno_podshipnika_EDT_1, err_mod:=arERR_3);
  AI_6_dblValue := arAIN_6.dblValue;

  (* [A1-5, AI1-0]  Т ОУП ЭД со стороны редуктора (т.2) *)
  fb_TOpornoYpornogoPodshipnikaEDT_2(arAIN := arAIN_7, strAI := ai.Toy_podshipnika_EDT_2, err_mod:=arERR_4);
  AI_7_dblValue := arAIN_7.dblValue;

  (* [A1-5, AI1-1]  Т ОУП колеса редуктора со стороны ЭД (т.3) *)
  fb_TOpornoYpornogoPodshipnikaKolesaRedEDT_3(arAIN := arAIN_8, strAI := ai.Toy_podshipnika_kol_EDT_3, err_mod:=arERR_4);
  AI_8_dblValue := arAIN_8.dblValue;

  (* [A1-5, AI1-2]Т ОП колеса редуктора со стороны Н (т.4) *)
  fb_TOpornoYpornogoPodshipnikaKolesaRedHT_4(arAIN := arAIN_9, strAI := ai.Toy_podshipnika_kol_EDT_4, err_mod:=arERR_4);
  AI_9_dblValue := arAIN_9.dblValue;

  (* [A1-5, AI1-3] Т ОП шестерни редуктора со стороны ЭД (т.5) *)
  fb_TOpornogoPodshipnikaShesterniReduktoraT_5(arAIN := arAIN_10, strAI := ai.Toy_podshipnika_shest_red_EDT_5, err_mod:=arERR_4);
  AI_10_dblValue := arAIN_10.dblValue;

  (* [A1-5, AI1-4]  Т ОП шестерни редуктора со стороны Н (т.6) *)
  fb_TOpornogoPodshipnikaReduktoraHT_6(arAIN := arAIN_11, strAI := ai.Ty_podshipnika_red_EDT_6, err_mod:=arERR_4);
  AI_11_dblValue := arAIN_11.dblValue;

  (* [A1-5, AI1-5]  Т ОП Н со стороны редуктора (т.7) *)
  fb_TOpornoYpornogoPodshipnikaNagnetateljaT_7_1(arAIN := arAIN_12, strAI := ai.Ty_podshipnika_nagnet_EDT_7_1, err_mod:=arERR_4);
  AI_12_dblValue := arAIN_12.dblValue;

  (* [A1-5, AI1-5]  Т ОП Н со стороны редуктора (т.7) *)
  fb_TOpornoYpornogoPodshipnikaNagnetateljaT_7_2(arAIN := arAIN_13, strAI := ai.Ty_podshipnika_nagnet_EDT_7_2, err_mod:=arERR_4);
  AI_13_dblValue := arAIN_13.dblValue;

  (* [A1-5, AI1-7]  Т ОП Н со стороны свободного вала (т.8) *)
  fb_TOpornoYpornogoPodshipnikaSvobodnogoKoncaNT_8_1(arAIN := arAIN_14, strAI := ai.Toy_podshipnika_svobod_konca_EDT_8_1, err_mod:=arERR_4);
  AI_14_dblValue := arAIN_14.dblValue;

  (* [A1-5, AI1-7]  Т ОП Н со стороны свободного вала (т.8) *)
  fb_TOpornoYpornogoPodshipnikaSvobodnogoKoncaNT_8_2(arAIN := arAIN_15, strAI := ai.Toy_podshipnika_svobod_konca_EDT_8_2, err_mod:=arERR_4);
  AI_15_dblValue := arAIN_15.dblValue;

  (* [A1-6, AI2-1]  Т УП рабочих колодок нагнетателя(т9) *)
  fb_TYpornogoPodshipnikaRabKolodokHT_9_1(arAIN := arAIN_16, strAI := ai.Toy_podshipnika_rab_kol_EDT_9_1, err_mod:=arERR_5);
  AI_16_dblValue := arAIN_16.dblValue;

  (* [A1-6, AI2-1]  Т УП рабочих колодок нагнетателя(т9) *)
  fb_TYpornogoPodshipnikaRabKolodokHT_9_2(arAIN := arAIN_17, strAI := ai.Toy_podshipnika_rab_kol_EDT_9_2, err_mod:=arERR_5);
  AI_17_dblValue := arAIN_17.dblValue;

  (* [A1-6, AI2-3]  Т ОП установочных колодок нагнетателя(т10) *)
  fb_TYpornogoPodshipnikYstanKolodokHT_10_1(arAIN := arAIN_18, strAI := ai.Toy_podshipnika_nerab_kol_EDT_10_1, err_mod:=arERR_5);
  AI_18_dblValue := arAIN_18.dblValue;

  (* [A1-6, AI2-3]  Т ОП установочных колодок нагнетателя(т10) *)
  fb_TYpornogoPodshipnikYstanKolodokHT_10_2(arAIN := arAIN_19, strAI := ai.Toy_podshipnika_nerab_kol_EDT_10_2, err_mod:=arERR_5);
  AI_19_dblValue := arAIN_19.dblValue;

  (* [A1-4, AI0-0] Т стали статора фаза 1 *)
  fb_TStalisStatoraKanal1(arAIN := arAIN_0, strAI := ai.Tstali_statora_kanal_1, err_mod:=arERR_3);
  AI_0_dblValue := arAIN_0.dblValue;

  (* [A1-4, AI0-1] Т стали статора фаза 2 *)
  fb_TStalisStatoraKanal2(arAIN := arAIN_1, strAI := ai.Tstali_statora_kanal_2, err_mod:=arERR_3);
  AI_1_dblValue := arAIN_1.dblValue;

  (* [A1-4, AI0-2] Т стали статора фаза 3 *)
  fb_TStalisStatoraKanal3(arAIN := arAIN_2, strAI := ai.Tstali_statora_kanal_3, err_mod:=arERR_3);
  AI_2_dblValue := arAIN_2.dblValue;

  (* [A1-6, AI2-5] Т холодного воздуха в ЭД, точка 1 *)
  fb_THolodnogoVozduhaEDKanall(arAIN := arAIN_20, strAI := ai.Tholodnogo_vozduha_ED_kanal_1, err_mod:=arERR_5);
  AI_20_dblValue := arAIN_20.dblValue;

  (* [A1-6, AI2-6] Т холодного воздуха в ЭД, точка 2 *)
  fb_THolodnogoVozduhaEDKanal2(arAIN := arAIN_21, strAI := ai.Tholodnogo_vozduha_ED_kanal_2, err_mod:=arERR_5);
  AI_21_dblValue := arAIN_21.dblValue;

  (* [A1-10, AI6-5] Уровень масла в маслобаке *)
  fb_YrovenMaslaMB(arAIN := arAIN_48, strAI := ai.Yroven_masla_MB, err_mod:=arERR_9);
  AI_48_dblValue := arAIN_48.dblValue;

  (* [A1-10, AI6-5] Уровень масла в маслобаке *)
  fb_VibroSkorostOPED_T1(arAIN := arAIN_56, strAI := ai.Kontrol_post_220V, err_mod:=arERR_9);
  AI_56_dblValue := arAIN_56.dblValue;

  (* [A1-10, AI6-5] Уровень масла в маслобаке *)
  fb_VibroSkorostOYPED_T2(arAIN := arAIN_57, strAI := ai.Vibro_skorost_OPED_T1, err_mod:=arERR_9);
  AI_57_dblValue := arAIN_57.dblValue;

  (* [A1-10, AI6-5] Уровень масла в маслобаке *)
  fb_VibroSkorostOPKolesaRH_T4(arAIN := arAIN_59, strAI := ai.Vibro_skorost_OP_kolesa_RH_T4, err_mod:=arERR_9);
  AI_59_dblValue := arAIN_59.dblValue;

  (* [A1-10, AI6-5] Уровень масла в маслобаке *)
  fb_VibroSkorostOPShesterniRED_T5(arAIN := arAIN_60, strAI := ai.Vibro_skorost_OP_shesterni_RED_T5, err_mod:=arERR_9);
  AI_60_dblValue := arAIN_60.dblValue;

  (* [A1-10, AI6-5] Уровень масла в маслобаке *)
  fb_VibroSkorostOPShesterniReduktoraH_T6(arAIN := arAIN_61, strAI := ai.Vibro_skorost_OP_shesterni_RED_T6, err_mod:=arERR_9);
  AI_61_dblValue := arAIN_61.dblValue;

  (**********************************************s Модуль A1-5 *********************************************************)
  A1_4_err_mode := arERR_3.wValue;
  A1_6_err_mode := arERR_5.wValue;
  A1_5_err_mode := arERR_4.wValue;
  A1_7_err_mode := arERR_6.wValue;

  (********************************************** Модуль A1-8 *********************************************************)
  (* [A1-8, AI4-5]  Температура в шкафу САУ *)
  fb_TEmperatura_v_SHU(arAIN := arAIN_32, strAI := ai.Tshu, err_mod:=arERR_7);
  AI_32_dblValue := arAIN_32.dblValue;

  (* [A1-9, AI5-5]  Вибрация ротора нагнетателя т.4 *)
  fb_OsSdvigNagnetatelja_Plus(arAIN := arAIN_42, strAI := ai.Os_sdvig_nagnetatelja_plus, err_mod:=arERR_8);
  AI_42_dblValue := arAIN_42.dblValue;

  (* [A1-9, AI5-6]  Осевой сдвиг ротора нагнетателя *)
  fb_OsSdvigNagnetatelja_Minus(arAIN := arAIN_43, strAI := ai.Os_sdvig_nagnetatelja_minus, err_mod:=arERR_8);
  AI_43_dblValue := arAIN_43.dblValue;

  A1_9_err_mode := arERR_8.wValue;

  (********************************************** Модуль A1-10 *********************************************************)
  (* [A1-10, AI6-0] Температура внутри шкафа *)
  fb_VibroSkorostOYPKolesaED_T3(arAIN := arAIN_58, strAI := ai.Vibro_skorost_OYP_kolesa_ED_T3, err_mod:=arERR_9);
  AI_58_dblValue := arAIN_58.dblValue;

  (* [A1-10, AI6-4] Активная мощность *)
  fb_DavlenieImpulsGaz(arAIN := arAIN_46, strAI := ai.Pimpuls_gaz, err_mod:=arERR_9);
  AI_46_dblValue := arAIN_46.dblValue;

  (* [A1-10, AI6-6]  Напряжение питания ШУ, основной ввод *)
  fb_Kontrol_per220V(arAIN := arAIN_52, strAI := ai.Kontrol_per_220V, err_mod:=arERR_9);
  AI_52_dblValue := arAIN_52.dblValue;

  (* [A1-10, AI6-7]  Напряжение питания ШУ, резервный ввод *)
  fb_Kontrol_post220V(arAIN := arAIN_53, strAI := ai.Kontrol_post_220V, err_mod:=arERR_9);
  AI_53_dblValue := arAIN_53.dblValue;

  (* [A1-10, AI6-7]  Напряжение питания ШУ, резервный ввод *)
  fb_TokStatora(arAIN := arAIN_65, strAI := ai.Tok_statora, err_mod:=arERR_9);
  AI_65_dblValue := arAIN_65.dblValue;

  A1_10_err_mode := arERR_9.wValue;
END_FUNCTION_BLOCK

FUNCTION_BLOCK Prov_K
  VAR_IN_OUT
    StrAlg : struct_Alg;
  END_VAR
  VAR
    F1_1_start : struct_PhaseAlgoritm;
    F1_2_start : struct_PhaseAlgoritm;
    F3_start : struct_PhaseAlgoritm;
    F4_Start : struct_PhaseAlgoritm;
    Start_Prov_Pusk : struct_Question;
    F4_Start_Q : struct_Question;
    fb_F1_1_start : fb_ph_algoritm;
    fb_F1_2_start : fb_ph_algoritm;
    fb_F3_start : fb_ph_algoritm;
    fb_F4_Start : fb_ph_Kran;
    algoritms : AlgoritmsConfig;
    fb_Start_Prov_Pusk : fb_Question;
    fb_F4_Start_Q : fb_Question;
    fb_kran4Open : fb_ph_Kran;
    fb_kran5Close : fb_ph_Kran;
    fb_kran4Close : fb_ph_Kran;
    fb_timer10 : fb_ph_Timer;
    fb_P_vh_vyh_more_zad : fb_ph_algoritm;
    fb_Zapoln_Norm : fb_ph_algoritm;
    fb_First_Step : fb_ph_algoritm;
    fb_Opressovka_Start : fb_Question;
    fb_PNS_NU_ON_Ask : fb_Question;
    fb_Zapolnit_kontur : fb_Question;
    onInit : BOOL;
  END_VAR
  VAR_EXTERNAL
    Im : ImConfig;
    ai : AiConfig;
  END_VAR
  VAR
    _sunpackerCommand : fb_sunpackerCommand;
    source : BYTE;
    cmd : BYTE;
    _statusDualInput : TYPE_statusDualInput;
    lastCmd : BYTE;
    _Answers : TYPE_Answers;
  END_VAR
  VAR_EXTERNAL
    ModeGpa : TYPE_ModeGpa;
    algManager : struct_AlgoritmsManager;
  END_VAR
  VAR
    cmd_for_Status : BYTE;
    source_for_Status : BYTE;
    command_error_for_Status : BYTE;
    resetCmdTimer : TON;
    waitReset : TON;
    resetCmdTimerPriznak : BOOL;
    _statusAi : TYPE_StatusAi;
    protections : ProtectionsConfig;
  END_VAR

  IF NOT onInit THEN
      fb_F1_1_start(phaseNumber:=1, act:=_run);
      fb_F1_2_start(phaseNumber:=2, act:=_run);
      fb_F3_start(phaseNumber:=3, act:=_run);
      fb_F4_Start(phaseNumber:=4, act:=_on);
      Start_Prov_Pusk.AnswerVariants:=_Answers.ANS_YES + _Answers.ANS_NO;
      F4_Start_Q.AnswerVariants:=_Answers.ANS_YES;
      onInit:=TRUE;
  END_IF;

  fb_F1_1_start(StrPh:=F1_1_start, alg := algoritms.Pusk_F_faza1);
  fb_F1_2_start(StrPh:=F1_2_start, alg := algoritms.Pusk_F_faza2);
  fb_F3_start(StrPh:=F3_start, alg := algoritms.Pusk_TH_faza);
  fb_F4_Start(StrPh:=F4_Start, Im:=Im.Kran6);
  fb_Start_Prov_Pusk(StrQ:=Start_Prov_Pusk);
  fb_F4_Start_Q(StrQ:=F4_Start_Q);

  StrAlg.CanRun := StrAlg.inCanRun;
  StrAlg.OpcCommandsDisabled := StrAlg.inOpcCommandsDisabled;

  IF StrAlg.isRuning THEN
      IF NOT F1_1_start.start THEN
  	askQuestion(Start_Prov_Pusk);
      END_IF;
      IF Start_Prov_Pusk.answer = _Answers.ANS_YES THEN
  	(*algoritms.F1_1.CanRun :=TRUE;*)
  	runPhase(F1_1_start);
  	resetQuestion(Start_Prov_Pusk);
  	(*algManager.setMode(nMode:=ModeGpa.MODE_PUSKK);*)
      ELSIF	Start_Prov_Pusk.answer=_Answers.ANS_NO THEN
  		resetQuestion(Start_Prov_Pusk);
  		(*algoritms.F1_1.CanRun :=FALSE;*)
      END_IF;
      IF F1_1_start.top THEN
  	(*algoritms.F1_2.CanRun :=TRUE;*)
  	runPhase(F1_2_start);
      END_IF;
      IF 	F1_2_start.top (*AND algoritms.ppu.ppuThird*)THEN
  	(*algoritms.F3.CanRun :=TRUE;*)
  	runPhase(F3_start);
      END_IF;
      IF F3_start.top AND (*algoritms.ppu.ppuForth AND*) NOT F4_Start.start  THEN
  	askQuestion(F4_Start_Q);
      ELSE
  	resetQuestion(F4_Start_Q);
      END_IF;
      IF F4_Start_Q.answer = _Answers.ANS_YES THEN
  	resetQuestion(F4_Start_Q);
  	(*algoritms.F4.CanRun :=TRUE;*)
  	runPhase(F4_Start);
      END_IF;
  END_IF;

  _sunpackerCommand(command := StrAlg.inCommand);
  	source := _sunpackerCommand.source;
  	cmd := _sunpackerCommand.cmd;

  IF cmd <> 0 AND lastCmd <> cmd AND (((NOT StrAlg.opcCommandsDisabled) AND source > 0) OR source = 0) then
  	CASE BYTE_TO_INT(cmd) OF
  		(*cm dRun*) 1: 	IF (StrAlg.CanRun) THEN
  					StrAlg.isRuning := TRUE;
  					StrAlg.isEnded := FALSE;
  					StrAlg.hasError := FALSE;
  					(*****************       OnRun       *****************)
                                                    algManager.nMode:=ModeGpa.MODE_PUSK_FIRST_FAZA2;

                                                    (*runPhase(timer120);
                                                    runPhase(timer5);
                                                    runPhase(Shup);
                                                    resetAiProtection(protections.dPmaslo_gaz);
                                                    resetDiProtection(protections.dPmaslo_gaz_less100);*)

  					cmd_for_Status := cmd;
  					source_for_Status := source;
  					command_error_for_Status := 0;
  				ELSE
  					StrAlg.isRuning := FALSE;
  					StrAlg.isEnded := FALSE;
  					StrAlg.hasError := FALSE;

  					cmd_for_Status := 0;
  					source_for_Status := source;
  					command_error_for_Status := cmd;
  				END_IF;
  		(*cmdReset*) 2: 	StrAlg.isRuning := FALSE;
  				StrAlg.isEnded := FALSE;
  				StrAlg.hasError 	:= FALSE;

                                           (*****************       OnReset       *****************)
                                          waitReset(IN:=FALSE);
                                          StrAlg.inCanRun:=FALSE;

                                          (*resetPhase(timer5);
                                          resetPhase(Shup);
                                          resetPhase(timer120);
                                          resetPhase(Net_Chast);
                                          resetPhase(mvOn);
                                          resetPhase(pGNSmore04);
                                          resetPhase(gotov_K_zagruzke);
                                          resetPhase(dPmg_Top);
                                          resetPhase(AutoPNS_Start);*)

                                          StrAlg.inOpcCommandsDisabled:=FALSE;

  				cmd_for_Status := cmd;
  				source_for_Status := source;
  				command_error_for_Status := 0;
  	END_CASE;
  	resetCmdTimer(IN := false);
  	resetCmdTimerPriznak := TRUE;
  END_IF;
  lastCmd := cmd;

  resetCmdTimer(IN := resetCmdTimerPriznak, PT := T#5S);
  IF resetCmdTimer.Q THEN
  	resetCmdTimerPriznak := FALSE;
  	source_for_Status := 0;
  	cmd_for_Status := 0;
  	command_error_for_Status := 0;
  END_IF;

  (*StrAlg.Start:= OPC_Control.startStatus
              OR Pms_more_50.startStatus
              OR Pms_more_300.startStatus
              OR dPmg_more_100.startStatus
              OR P_zad.startStatus
              OR kran5Open.startStatus
              OR kran4Open.startStatus
              OR kran5Close.startStatus
              OR kran4Close.startStatus
              OR timer10.startStatus
              OR P_vh_vyh_more_zad.startStatus
              OR Zapoln_Norm.startStatus
              OR First_Step.startStatus;

  StrAlg.Top :=  OPC_Control.topStatus
              OR Pms_more_50.topStatus
              OR Pms_more_300.topStatus
              OR dPmg_more_100.topStatus
              OR P_zad.topStatus
              OR kran5Open.topStatus
              OR kran4Open.topStatus
              OR kran5Close.topStatus
              OR kran4Close.topStatus
              OR timer10.topStatus
              OR P_vh_vyh_more_zad.topStatus
              OR Zapoln_Norm.topStatus
              OR First_Step.topStatus;

  StrAlg.Error :=  OPC_Control.errorStatus
              OR Pms_more_50.errorStatus
              OR Pms_more_300.errorStatus
              OR dPmg_more_100.errorStatus
              OR P_zad.errorStatus
              OR kran5Open.errorStatus
              OR kran4Open.errorStatus
              OR kran5Close.errorStatus
              OR kran4Close.errorStatus
              OR timer10.errorStatus
              OR P_vh_vyh_more_zad.errorStatus
              OR Zapoln_Norm.errorStatus
              OR First_Step.errorStatus;*)

  (*TODO: TYPE PROGRAM CODE HERE*)
  StrAlg.status :=  SHL(BYTE_TO_DWORD(source_for_Status), 29)
  			OR SHL(BYTE_TO_DWORD(cmd_for_Status), 26)
  			OR SHL(BYTE_TO_DWORD(command_error_for_Status), 23)
  			OR SHL(BOOL_TO_DWORD(StrAlg.OpcCommandsDisabled ), 21)
  			OR SHL(BOOL_TO_DWORD(StrAlg.hasError),4)
  			OR SHL(BOOL_TO_DWORD(StrAlg.CanRun),2)
  			OR SHL(BOOL_TO_DWORD(StrAlg.isEnded),1)
  			OR BOOL_TO_DWORD(StrAlg.isRuning);
END_FUNCTION_BLOCK

FUNCTION_BLOCK Prov_dP_mg
  VAR_IN_OUT
    StrAlg : struct_Alg;
  END_VAR
  VAR
    nu1Off : struct_PhaseAlgoritm;
    nu2Off : struct_PhaseAlgoritm;
    pnsOff : struct_PhaseAlgoritm;
    timer120 : struct_PhaseAlgoritm;
    dPmg_less_100 : struct_PhaseAlgoritm;
    nu1On : struct_PhaseAlgoritm;
    nu2On : struct_PhaseAlgoritm;
    pnsOn : struct_PhaseAlgoritm;
    Error_Alg : struct_PhaseAlgoritm;
    dPmg_more_100 : struct_PhaseAlgoritm;
    fb_nu1Off : fb_ph_OilPump;
    fb_nu2Off : fb_ph_OilPump;
    fb_pnsOff : fb_ph_Switch;
    fb_timer120 : fb_ph_Timer;
    fb_dPmg_less_100 : fb_ph_algoritm;
    fb_nu1On : fb_ph_OilPump;
    fb_nu2On : fb_ph_OilPump;
    fb_pnsOn : fb_ph_Switch;
    fb_Error_Alg : fb_ph_algoritm;
    fb_dPmg_more_100 : fb_ph_algoritm;
    onInit : BOOL;
  END_VAR
  VAR_EXTERNAL
    Im : ImConfig;
    ai : AiConfig;
  END_VAR
  VAR
    _sunpackerCommand : fb_sunpackerCommand;
    source : BYTE;
    cmd : BYTE;
    _statusDualInput : TYPE_statusDualInput;
    lastCmd : BYTE;
    _Answers : TYPE_Answers;
  END_VAR
  VAR_EXTERNAL
    ModeGpa : TYPE_ModeGpa;
    algManager : struct_AlgoritmsManager;
  END_VAR
  VAR
    cmd_for_Status : BYTE;
    source_for_Status : BYTE;
    command_error_for_Status : BYTE;
    resetCmdTimer : TON;
    waitReset : TON;
    resetCmdTimerPriznak : BOOL;
  END_VAR

  IF NOT onInit THEN
      fb_nu1Off(phaseNumber:=1, act:=_off);
      fb_nu2Off(phaseNumber:=2, act:=_off);
      fb_pnsOff(phaseNumber:=3, act:=_off);
      fb_timer120(phaseNumber:=4, delay:=T#120S);
      fb_dPmg_less_100(phaseNumber:=5);
      fb_nu1On(phaseNumber:=6, act:=_on);
      fb_nu2On(phaseNumber:=7, act:=_on);
      fb_pnsOn(phaseNumber:=8, act:=_on);
      fb_Error_Alg(phaseNumber:=9);
      fb_dPmg_more_100(phaseNumber:=10);
      onInit:=TRUE;
  END_IF;

  fb_nu1Off(StrPh:=nu1Off, Im:=Im.nu1);
  fb_nu2Off(StrPh:=nu2Off, Im:=Im.nu2);
  fb_pnsOff(StrPh:=pnsOff, Im:=Im.pns);
  fb_timer120(StrPh:=timer120);
  fb_dPmg_less_100(StrPh:=dPmg_less_100);
  fb_nu1On(StrPh:=nu1On, Im:=Im.nu1);
  fb_nu2On(StrPh:=nu2On, Im:=Im.nu2);
  fb_pnsOn(StrPh:=pnsOn, Im:=Im.pns);
  fb_Error_Alg(StrPh:=Error_Alg);
  fb_dPmg_more_100(StrPh:=dPmg_more_100);

  StrAlg.CanRun := StrAlg.inCanRun;
  StrAlg.OpcCommandsDisabled := StrAlg.inOpcCommandsDisabled;

      IF StrAlg.isRuning THEN
      (* kto takoi ask
          IF	NOT nuOff.start THEN
  	    NU_OFF_Ask.ask ();
      END_IF;*)

      (*
      IF	(nu_OFF_Ask.answer=Answers.ANS_YES) THEN
  	    runPhase(nu1Off);
  	    runPhase(nu2Off);
          runPhase(pnsOff);
  	    NU_OFF_Ask.reset ();
  	    runPhase(timer120);
      END_IF;*)

      (*насосы выключены - запуск проверки *)
      IF	nu1Off.top AND nu2Off.top THEN
  	    runPhase(dPmg_less_100);
      END_IF;

      (*проверка перепада маслогаз по аналогу и дискрету*)
      IF	dPmg_less_100.start AND NOT dPmg_less_100.top THEN
          IF 	Im.SingleSignals.dP_maslo_gaz_Less100.Q AND ai.dPmaslo_gaz.value < 150.0 THEN
  	  	    dPmg_less_100.top:=TRUE;
  		    runPhase(nu1On);
              runPhase(nu2On);
              runPhase(pnsOn);
  	    END_IF;
      END_IF;

      IF	Im.nu1.onStatus = _statusDualInput.STATUS_ON OR Im.nu2.onStatus = _statusDualInput.STATUS_ON  AND nu1On.start  AND nu2On.start AND NOT nu1On.top AND NOT nu2On.top THEN
  	    nu1On.top := TRUE;
          nu2On.top := TRUE;
      END_IF;

      (*ошибка завершения по таймеру*)
      IF	timer120.top THEN
  	    Error_Alg.ERROR := TRUE;
      ELSE
  	    Error_Alg.ERROR := FALSE;
      END_IF;

      (*ыва*)
      IF	nu1On.top AND nu2On.top AND pnsOn.top THEN
  	    runPhase(dPmg_more_100);
      END_IF;

      (**)
      IF	dPmg_more_100.start AND NOT dPmg_more_100.top (*AND NOT algoritms.autoNu_1.flag1 OR algoritms.autoNu_1.flag2*) THEN
  	    IF 	NOT Im.SingleSignals.dP_maslo_gaz_Less100.Q AND Im.SingleSignals.dP_maslo_gaz_Less100.status = 1 AND  ai.dPmaslo_gaz.value > 150.0 THEN
      		dPmg_more_100.top :=TRUE;
  		    resetPhase(timer120);
  	    END_IF;
      END_IF;
  END_IF;

  _sunpackerCommand(command := StrAlg.inCommand);
  	source := _sunpackerCommand.source;
  	cmd := _sunpackerCommand.cmd;

  IF cmd <> 0 AND lastCmd <> cmd AND (((NOT StrAlg.opcCommandsDisabled) AND source > 0) OR source = 0) then
  	CASE BYTE_TO_INT(cmd) OF
  		(*cm dRun*) 1: 	IF (StrAlg.CanRun) THEN
  					StrAlg.isRuning := TRUE;
  					StrAlg.isEnded := FALSE;
  					StrAlg.hasError := FALSE;
  					(*****************       OnRun       *****************)
                                                    algManager.nMode:=ModeGpa.MODE_PUSK_FIRST_FAZA2;

                                                    (*runPhase(timer120);
                                                    runPhase(timer5);
                                                    runPhase(Shup);
                                                    resetAiProtection(protections.dPmaslo_gaz);
                                                    resetDiProtection(protections.dPmaslo_gaz_less100);*)

  					cmd_for_Status := cmd;
  					source_for_Status := source;
  					command_error_for_Status := 0;
  				ELSE
  					StrAlg.isRuning := FALSE;
  					StrAlg.isEnded := FALSE;
  					StrAlg.hasError := FALSE;

  					cmd_for_Status := 0;
  					source_for_Status := source;
  					command_error_for_Status := cmd;
  				END_IF;
  		(*cmdReset*) 2: 	StrAlg.isRuning := FALSE;
  				StrAlg.isEnded := FALSE;
  				StrAlg.hasError 	:= FALSE;

                                           (*****************       OnReset       *****************)
                                          waitReset(IN:=FALSE);
                                          StrAlg.inCanRun:=FALSE;

                                          (*resetPhase(timer5);
                                          resetPhase(Shup);
                                          resetPhase(timer120);
                                          resetPhase(Net_Chast);
                                          resetPhase(mvOn);
                                          resetPhase(pGNSmore04);
                                          resetPhase(gotov_K_zagruzke);
                                          resetPhase(dPmg_Top);
                                          resetPhase(AutoPNS_Start);*)

                                          StrAlg.inOpcCommandsDisabled:=FALSE;

  				cmd_for_Status := cmd;
  				source_for_Status := source;
  				command_error_for_Status := 0;
  	END_CASE;
  	resetCmdTimer(IN := false);
  	resetCmdTimerPriznak := TRUE;
  END_IF;
  lastCmd := cmd;

  resetCmdTimer(IN := resetCmdTimerPriznak, PT := T#5S);
  IF resetCmdTimer.Q THEN
  	resetCmdTimerPriznak := FALSE;
  	source_for_Status := 0;
  	cmd_for_Status := 0;
  	command_error_for_Status := 0;
  END_IF;

  StrAlg.Start:= nu1Off.startStatus
              OR nu2Off.startStatus
              OR pnsOff.startStatus
              OR timer120.startStatus
              OR dPmg_less_100.startStatus
              OR nu1On.startStatus
              OR nu2On.startStatus
              OR pnsOn.startStatus;

  StrAlg.Top := nu1Off.topStatus
              OR nu2Off.topStatus
              OR pnsOff.topStatus
              OR timer120.topStatus
              OR dPmg_less_100.topStatus
              OR nu1On.topStatus
              OR nu2On.topStatus
              OR pnsOn.topStatus;

  StrAlg.Error := nu1Off.errorStatus
              OR nu2Off.errorStatus
              OR pnsOff.errorStatus
              OR timer120.errorStatus
              OR dPmg_less_100.errorStatus
              OR nu1On.errorStatus
              OR nu2On.errorStatus
              OR pnsOn.errorStatus;

  (*TODO: TYPE PROGRAM CODE HERE*)
  StrAlg.status :=  SHL(BYTE_TO_DWORD(source_for_Status), 29)
  			OR SHL(BYTE_TO_DWORD(cmd_for_Status), 26)
  			OR SHL(BYTE_TO_DWORD(command_error_for_Status), 23)
  			OR SHL(BOOL_TO_DWORD(StrAlg.OpcCommandsDisabled ), 21)
  			OR SHL(BOOL_TO_DWORD(StrAlg.hasError),4)
  			OR SHL(BOOL_TO_DWORD(StrAlg.CanRun),2)
  			OR SHL(BOOL_TO_DWORD(StrAlg.isEnded),1)
  			OR BOOL_TO_DWORD(StrAlg.isRuning);
END_FUNCTION_BLOCK

FUNCTION_BLOCK fb_DiProtection_Init
  VAR_INPUT
    data_Ini : BOOL;
    delay : TIME;
    inTag : BYTE;
    inRunOnStart : BOOL;
  END_VAR
  VAR_IN_OUT
    str_DIp : struct_DiProtection;
  END_VAR
  VAR_OUTPUT
    Init : BOOL      := FALSE;
  END_VAR

  (*****            Функциональный блок переинициализации структуры  AiProtection          *****)

   Init := FALSE;

      IF data_Ini THEN                            (* Параметрам требуется переинициализация. *)
          str_DIp.delay               := delay;
          str_DIp.inTag               := inTag;
          str_DIp.inRunOnStart        := inRunOnStart;

          data_Ini:=FALSE;
          Init := TRUE;
      END_IF;
      IF Init THEN
          delay:= T#0S;
          inTag:= 0;
          inRunOnStart:= FALSE;
      END_IF;
END_FUNCTION_BLOCK

FUNCTION_BLOCK proc_Protections_Init
  VAR_INPUT
    init : BOOL;
  END_VAR
  VAR
    stDIp_Ini : fb_DiProtection_Init;
    stAIp_Ini : fb_AiProtection_Init;
    inits : UINT;
  END_VAR
  VAR_INPUT
    initiales : UINT;
  END_VAR
  VAR_EXTERNAL
    protections : ProtectionsConfig;
  END_VAR
  VAR
    _ProtectionTags : TYPE_ProtectionTags;
    _StatusAi : TYPE_StatusAi;
  END_VAR

  inits := 0; (* Флаг необходимости инициализации структур-дескрипторов *)

  (*************************************************Стартовая инициализация DiProtection ***************************************************)
  (* МВ отключен *)
  stDIp_Ini(data_Ini := true, delay:=T#03S, inTag:=_ProtectionTags.AOS, inRunOnStart:=TRUE, str_DIp := protections.Reg_vozb_off);
  inits := inits + BOOL_TO_UINT(stDIp_Ini.Init);

  (* МВ отключен
  stDIp_Ini(data_Ini := true, delay:=T#1S, inTag:=_ProtectionTags.AOS, inRunOnStart:=FALSE, str_DIp := protections.Fail_chastotnii_pusk);
  inits := inits + BOOL_TO_UINT(stDIp_Ini.Init);*)

  (* МВ отключен *)
  stDIp_Ini(data_Ini := true, delay:=T#1S, inTag:=_ProtectionTags.AOS, inRunOnStart:=TRUE, str_DIp := protections.Off_avar_vikluchatel);
  inits := inits + BOOL_TO_UINT(stDIp_Ini.Init);

  (* МВ отключен *)
  stDIp_Ini(data_Ini := true, delay:=T#1S, inTag:=_ProtectionTags.AOS, inRunOnStart:=TRUE, str_DIp := protections.AOKC_SHKC);
  inits := inits + BOOL_TO_UINT(stDIp_Ini.Init);

  (* МВ отключен *)
  stDIp_Ini(data_Ini := true, delay:=T#0S, inTag:=_ProtectionTags.AOS, inRunOnStart:=TRUE, str_DIp := protections.AO_PRU);
  inits := inits + BOOL_TO_UINT(stDIp_Ini.Init);

  (* МВ отключен *)
  stDIp_Ini(data_Ini := true, delay:=T#0S, inTag:=_ProtectionTags.AOS, inRunOnStart:=FALSE, str_DIp := protections.AO_ot_SHU);
  inits := inits + BOOL_TO_UINT(stDIp_Ini.Init);

  (* МВ отключен *)
  stDIp_Ini(data_Ini := true, delay:=T#1S, inTag:=_ProtectionTags.AOS, inRunOnStart:=FALSE, str_DIp := protections.mvOff);
  inits := inits + BOOL_TO_UINT(stDIp_Ini.Init);

  (* МВ отключен *)
  stDIp_Ini(data_Ini := true, delay:=T#10S, inTag:=_ProtectionTags.AOS, inRunOnStart:=TRUE, str_DIp := protections.Kran1_sdvig);
  inits := inits + BOOL_TO_UINT(stDIp_Ini.Init);

  (* МВ отключен *)
  stDIp_Ini(data_Ini := true, delay:=T#10S, inTag:=_ProtectionTags.AOS, inRunOnStart:=TRUE, str_DIp := protections.Kran2_sdvig);
  inits := inits + BOOL_TO_UINT(stDIp_Ini.Init);

  (* МВ отключен *)
  stDIp_Ini(data_Ini := true, delay:=T#20S, inTag:=_ProtectionTags.AOS, inRunOnStart:=TRUE, str_DIp := protections.dPmaslo_gaz_less100);
  inits := inits + BOOL_TO_UINT(stDIp_Ini.Init);

  (*************************************************Стартовая инициализация AiProtection ***************************************************)
  (* Температура переднего опорного подшипника двигателя, т.1 *)
  stAIp_Ini(data_Ini := true, delay:=T#3S, inTag:=_ProtectionTags.AOS, inRunOnStart:=TRUE,
  controlLimit:=_StatusAi.HA, str_AIp := protections.Topornogo_podshipnika_EDT_1);
  inits := inits + BOOL_TO_UINT(stAIp_Ini.Init);

  (* Температура заднего опорного подшипника двигателя, т.2 *)
  stAIp_Ini(data_Ini := true, delay:=T#3S, inTag:=_ProtectionTags.AOS, inRunOnStart:=TRUE,
  controlLimit:=_StatusAi.HA, str_AIp := protections.Toy_podshipnika_EDT_2);
  inits := inits + BOOL_TO_UINT(stAIp_Ini.Init);

  (* Температура подшипника редуктора, т1 *)
  stAIp_Ini(data_Ini := true, delay:=T#3S, inTag:=_ProtectionTags.AOS, inRunOnStart:=TRUE,
  controlLimit:=_StatusAi.HA, str_AIp := protections.Toy_podshipnika_kol_EDT_3);
  inits := inits + BOOL_TO_UINT(stAIp_Ini.Init);

  (* Температура подшипника редуктора, т2 *)
  stAIp_Ini(data_Ini := true, delay:=T#3S, inTag:=_ProtectionTags.AOS, inRunOnStart:=TRUE,
  controlLimit:=_StatusAi.HA, str_AIp := protections.Toy_podshipnika_kol_EDT_4);
  inits := inits + BOOL_TO_UINT(stAIp_Ini.Init);

  (* Температура подшипника редуктора, т3 *)
  stAIp_Ini(data_Ini := true, delay:=T#3S, inTag:=_ProtectionTags.AOS, inRunOnStart:=TRUE,
  controlLimit:=_StatusAi.HA, str_AIp := protections.To_podshipnika_shest_red_EDT_5);
  inits := inits + BOOL_TO_UINT(stAIp_Ini.Init);

  (* Температура подшипника редуктора, т4 *)
  stAIp_Ini(data_Ini := true, delay:=T#3S, inTag:=_ProtectionTags.AOS, inRunOnStart:=TRUE,
  controlLimit:=_StatusAi.HA, str_AIp := protections.To_podshipnika_shest_red_EDT_6);
  inits := inits + BOOL_TO_UINT(stAIp_Ini.Init);

  (* Температура опорного подшипника нагнетателя, т1 *)
  stAIp_Ini(data_Ini := true, delay:=T#3S, inTag:=_ProtectionTags.AOS, inRunOnStart:=TRUE,
  controlLimit:=_StatusAi.HA, str_AIp := protections.To_podshipnika_N_EDT_7);
  inits := inits + BOOL_TO_UINT(stAIp_Ini.Init);

  (* Температура опорного подшипника нагнетателя, т2 *)
  stAIp_Ini(data_Ini := true, delay:=T#3S, inTag:=_ProtectionTags.AOS, inRunOnStart:=TRUE,
  controlLimit:=_StatusAi.HA, str_AIp := protections.To_podshipnika_svob_konca_EDT_8);
  inits := inits + BOOL_TO_UINT(stAIp_Ini.Init);

  (* Температура опорного подшипника нагнетателя, т3 *)
  stAIp_Ini(data_Ini := true, delay:=T#3S, inTag:=_ProtectionTags.AOS, inRunOnStart:=TRUE,
  controlLimit:=_StatusAi.HA, str_AIp := protections.Ty_podshipnika_rab_kol_EDT_9);
  inits := inits + BOOL_TO_UINT(stAIp_Ini.Init);

  (* Температура упорно опорного подшипника нагнетателя, т4 *)
  stAIp_Ini(data_Ini := true, delay:=T#3S, inTag:=_ProtectionTags.AOS, inRunOnStart:=TRUE,
  controlLimit:=_StatusAi.HA, str_AIp := protections.Typornogo_podshipnika_nerab_kolodok_HT_10);
  inits := inits + BOOL_TO_UINT(stAIp_Ini.Init);

  (* Температура газа на выходе нагнетателя *)
  stAIp_Ini(data_Ini := true, delay:=T#3S, inTag:=_ProtectionTags.AOS, inRunOnStart:=TRUE,
  controlLimit:=_StatusAi.HA, str_AIp := protections.Tgaza_na_vyhode_H);
  inits := inits + BOOL_TO_UINT(stAIp_Ini.Init);

  (* Температура газа на выходе нагнетателя *)
  stAIp_Ini(data_Ini := true, delay:=T#3S, inTag:=_ProtectionTags.AOS, inRunOnStart:=TRUE,
  controlLimit:=_StatusAi.HA, str_AIp := protections.Os_sdvig_nagnetatelja_plus);
  inits := inits + BOOL_TO_UINT(stAIp_Ini.Init);

  (* Температура газа на выходе нагнетателя *)
  stAIp_Ini(data_Ini := true, delay:=T#3S, inTag:=_ProtectionTags.AOS, inRunOnStart:=TRUE,
  controlLimit:=_StatusAi.HA, str_AIp := protections.Os_sdvig_nagnetatelja_minus);
  inits := inits + BOOL_TO_UINT(stAIp_Ini.Init);

  (* Температура газа на выходе нагнетателя *)
  stAIp_Ini(data_Ini := true, delay:=T#3S, inTag:=_ProtectionTags.AOS, inRunOnStart:=TRUE,
  controlLimit:=_StatusAi.HA, str_AIp := protections.Pgaza_na_vyhode_nagnetatelia_GPA_STOP);
  inits := inits + BOOL_TO_UINT(stAIp_Ini.Init);

  (* Температура газа на выходе нагнетателя *)
  stAIp_Ini(data_Ini := true, delay:=T#3S, inTag:=_ProtectionTags.AOS, inRunOnStart:=TRUE,
  controlLimit:=_StatusAi.HA, str_AIp := protections.Pgaza_na_vhode_nagnetatelia_GPA_STOP);
  inits := inits + BOOL_TO_UINT(stAIp_Ini.Init);

  (* Температура газа на выходе нагнетателя *)
  stAIp_Ini(data_Ini := true, delay:=T#3S, inTag:=_ProtectionTags.AOS, inRunOnStart:=TRUE,
  controlLimit:=_StatusAi.HA, str_AIp := protections.Pgaza_na_vyhode_nagnetatelia);
  inits := inits + BOOL_TO_UINT(stAIp_Ini.Init);

  (* Температура газа на выходе нагнетателя *)
  stAIp_Ini(data_Ini := true, delay:=T#20S, inTag:=_ProtectionTags.AOS, inRunOnStart:=TRUE,
  controlLimit:=_StatusAi.HA, str_AIp := protections.dPmaslo_gaz);
  inits := inits + BOOL_TO_UINT(stAIp_Ini.Init);

  (* Температура газа на выходе нагнетателя *)
  stAIp_Ini(data_Ini := true, delay:=T#16S, inTag:=_ProtectionTags.AOS, inRunOnStart:=TRUE,
  controlLimit:=_StatusAi.HA, str_AIp := protections.Pmaslo_sm_nizkoe);
  inits := inits + BOOL_TO_UINT(stAIp_Ini.Init);

  (* Температура газа на выходе нагнетателя *)
  stAIp_Ini(data_Ini := true, delay:=T#16S, inTag:=_ProtectionTags.AOS, inRunOnStart:=TRUE,
  controlLimit:=_StatusAi.HA, str_AIp := protections.Pmaslo_sm_vysokoe);
  inits := inits + BOOL_TO_UINT(stAIp_Ini.Init);

   (* Температура газа на выходе нагнетателя *)
  stAIp_Ini(data_Ini := true, delay:=T#3S, inTag:=_ProtectionTags.AOS, inRunOnStart:=TRUE,
  controlLimit:=_StatusAi.HA, str_AIp := protections.Vibro_skorost_OPED_T1);
  inits := inits + BOOL_TO_UINT(stAIp_Ini.Init);

   (* Температура газа на выходе нагнетателя *)
  stAIp_Ini(data_Ini := true, delay:=T#3S, inTag:=_ProtectionTags.AOS, inRunOnStart:=TRUE,
  controlLimit:=_StatusAi.HA, str_AIp := protections.Vibro_skorost_OPED_T2);
  inits := inits + BOOL_TO_UINT(stAIp_Ini.Init);

   (* Температура газа на выходе нагнетателя *)
  stAIp_Ini(data_Ini := true, delay:=T#3S, inTag:=_ProtectionTags.AOS, inRunOnStart:=TRUE,
  controlLimit:=_StatusAi.HA, str_AIp := protections.Vibro_skorost_OYP_kolesa_ED_T3);
  inits := inits + BOOL_TO_UINT(stAIp_Ini.Init);

   (* Температура газа на выходе нагнетателя *)
  stAIp_Ini(data_Ini := true, delay:=T#3S, inTag:=_ProtectionTags.AOS, inRunOnStart:=TRUE,
  controlLimit:=_StatusAi.HA, str_AIp := protections.Vibro_skorost_OP_kolesa_RH_T4);
  inits := inits + BOOL_TO_UINT(stAIp_Ini.Init);

   (* Температура газа на выходе нагнетателя *)
  stAIp_Ini(data_Ini := true, delay:=T#3S, inTag:=_ProtectionTags.AOS, inRunOnStart:=TRUE,
  controlLimit:=_StatusAi.HA, str_AIp := protections.Vibro_skorost_OP_shesterni_RED_T5);
  inits := inits + BOOL_TO_UINT(stAIp_Ini.Init);

   (* Температура газа на выходе нагнетателя *)
  stAIp_Ini(data_Ini := true, delay:=T#3S, inTag:=_ProtectionTags.AOS, inRunOnStart:=TRUE,
  controlLimit:=_StatusAi.HA, str_AIp := protections.Vibro_skorost_OP_shesterni_RED_T6);
  inits := inits + BOOL_TO_UINT(stAIp_Ini.Init);

   (* Температура газа на выходе нагнетателя *)
  stAIp_Ini(data_Ini := true, delay:=T#3S, inTag:=_ProtectionTags.AOS, inRunOnStart:=TRUE,
  controlLimit:=_StatusAi.HA, str_AIp := protections.Vibro_skorost_OYP_kolesa_ED_T3);
  inits := inits + BOOL_TO_UINT(stAIp_Ini.Init);

   (* Температура газа на выходе нагнетателя *)
  stAIp_Ini(data_Ini := true, delay:=T#3S, inTag:=_ProtectionTags.AOS, inRunOnStart:=TRUE,
  controlLimit:=_StatusAi.HA, str_AIp := protections.Vibro_skorost_OYP_kolesa_ED_T3);
  inits := inits + BOOL_TO_UINT(stAIp_Ini.Init);

   (* Температура газа на выходе нагнетателя *)
  stAIp_Ini(data_Ini := true, delay:=T#3S, inTag:=_ProtectionTags.AOS, inRunOnStart:=TRUE,
  controlLimit:=_StatusAi.HA, str_AIp := protections.Vibro_skorost_OYP_kolesa_ED_T3);
  inits := inits + BOOL_TO_UINT(stAIp_Ini.Init);

  IF init THEN initiales := inits; END_IF;
END_FUNCTION_BLOCK

FUNCTION runAllProtections : BOOL
  VAR_IN_OUT
    protections : ProtectionsConfig;
  END_VAR

  runAiProtection(protections.Topornogo_podshipnika_EDT_1);
  runAiProtection(protections.Toy_podshipnika_EDT_2);
  runAiProtection(protections.Toy_podshipnika_kol_EDT_3);
  runAiProtection(protections.Toy_podshipnika_kol_EDT_4);
  runAiProtection(protections.To_podshipnika_shest_red_EDT_5);
  runAiProtection(protections.To_podshipnika_shest_red_EDT_6);
  runAiProtection(protections.To_podshipnika_N_EDT_7);
  runAiProtection(protections.To_podshipnika_svob_konca_EDT_8);
  runAiProtection(protections.Ty_podshipnika_rab_kol_EDT_9);
  runAiProtection(protections.Typornogo_podshipnika_nerab_kolodok_HT_10);
  runAiProtection(protections.Tgaza_na_vyhode_H);
  runAiProtection(protections.Os_sdvig_nagnetatelja_plus);
  runAiProtection(protections.Os_sdvig_nagnetatelja_minus);
  runAiProtection(protections.Pgaza_na_vyhode_nagnetatelia_GPA_STOP);
  runAiProtection(protections.Pgaza_na_vhode_nagnetatelia_GPA_STOP);
  runAiProtection(protections.Pgaza_na_vyhode_nagnetatelia);
  runAiProtection(protections.dPmaslo_gaz);
  runAiProtection(protections.Pmaslo_sm_nizkoe);
  runAiProtection(protections.Pmaslo_sm_vysokoe);
  runAiProtection(protections.Vibro_skorost_OPED_T1);
  runAiProtection(protections.Vibro_skorost_OPED_T2);
  runAiProtection(protections.Vibro_skorost_OYP_kolesa_ED_T3);
  runAiProtection(protections.Vibro_skorost_OP_kolesa_RH_T4);
  runAiProtection(protections.Vibro_skorost_OP_shesterni_RED_T5);
  runAiProtection(protections.Vibro_skorost_OP_shesterni_RED_T6);

  runDiProtection(protections.dPmaslo_gaz_less100);
  runDiProtection(protections.Reg_vozb_off);
  runDiProtection(protections.Fail_chastotnii_pusk);
  runDiProtection(protections.Off_avar_vikluchatel);
  runDiProtection(protections.AOKC_SHKC);
  runDiProtection(protections.AO_PRU);
  runDiProtection(protections.AO_ot_SHU);
  runDiProtection(protections.mvOff);
  runDiProtection(protections.Kran1_sdvig);
  runDiProtection(protections.Kran2_sdvig);
END_FUNCTION

FUNCTION autoRunProtections : BOOL
  VAR_IN_OUT
    protections : ProtectionsConfig;
  END_VAR

  runAiProtection(protections.Topornogo_podshipnika_EDT_1);

      runAiProtection(protections.Toy_podshipnika_EDT_2);

      runAiProtection(protections.Toy_podshipnika_kol_EDT_3);

      runAiProtection(protections.Toy_podshipnika_kol_EDT_4);

      runAiProtection(protections.To_podshipnika_shest_red_EDT_5);

      runAiProtection(protections.To_podshipnika_shest_red_EDT_6);

      runAiProtection(protections.To_podshipnika_N_EDT_7);

      runAiProtection(protections.To_podshipnika_svob_konca_EDT_8);

      runAiProtection(protections.Ty_podshipnika_rab_kol_EDT_9);

      runAiProtection(protections.Typornogo_podshipnika_nerab_kolodok_HT_10);

      runAiProtection(protections.Tgaza_na_vyhode_H);

      runAiProtection(protections.Os_sdvig_nagnetatelja_plus);

      runAiProtection(protections.Os_sdvig_nagnetatelja_minus);

      runAiProtection(protections.Pgaza_na_vyhode_nagnetatelia_GPA_STOP);

      runAiProtection(protections.Pgaza_na_vhode_nagnetatelia_GPA_STOP);

      runAiProtection(protections.Pgaza_na_vyhode_nagnetatelia);

      runAiProtection(protections.dPmaslo_gaz);

      runAiProtection(protections.Pmaslo_sm_nizkoe);

      runAiProtection(protections.Pmaslo_sm_vysokoe);

      runAiProtection(protections.Vibro_skorost_OPED_T1);

      runAiProtection(protections.Vibro_skorost_OPED_T2);

      runAiProtection(protections.Vibro_skorost_OYP_kolesa_ED_T3);

      runAiProtection(protections.Vibro_skorost_OP_kolesa_RH_T4);

      runAiProtection(protections.Vibro_skorost_OP_shesterni_RED_T5);

      runAiProtection(protections.Vibro_skorost_OP_shesterni_RED_T6);

      runDiProtection(protections.dPmaslo_gaz_less100);

      runDiProtection(protections.AO_PRU);

      runDiProtection(protections.Reg_vozb_off);

      runDiProtection(protections.Fail_chastotnii_pusk);

      runDiProtection(protections.AOKC_SHKC);

      runDiProtection(protections.mvOff);

      runDiProtection(protections.AO_ot_SHU);

      runDiProtection(protections.Off_avar_vikluchatel);

      runDiProtection(protections.Kran1_sdvig);

      runDiProtection(protections.Kran2_sdvig);
END_FUNCTION

FUNCTION anyProtectionInRemont : BOOL
  VAR_INPUT
    protections : ProtectionsConfig;
  END_VAR

  anyProtectioninRemont:=
  protections.Topornogo_podshipnika_EDT_1.Remont OR
  protections.Toy_podshipnika_EDT_2.Remont OR
  protections.Toy_podshipnika_kol_EDT_3.remont OR
  protections.Toy_podshipnika_kol_EDT_4.Remont OR
  protections.To_podshipnika_shest_red_EDT_5.Remont OR
  protections.To_podshipnika_shest_red_EDT_6.Remont OR
  protections.To_podshipnika_N_EDT_7.Remont OR
  protections.To_podshipnika_svob_konca_EDT_8.Remont OR
  protections.Ty_podshipnika_rab_kol_EDT_9.Remont OR
  protections.Typornogo_podshipnika_nerab_kolodok_HT_10.Remont OR
  protections.Tgaza_na_vyhode_H.Remont OR
  protections.Os_sdvig_nagnetatelja_plus.Remont OR
  protections.Os_sdvig_nagnetatelja_minus.Remont OR
  protections.Pgaza_na_vyhode_nagnetatelia_GPA_STOP.Remont OR
  protections.Pgaza_na_vhode_nagnetatelia_GPA_STOP.Remont OR
  protections.Pgaza_na_vyhode_nagnetatelia.Remont OR
  protections.dPmaslo_gaz.Remont OR
  protections.Pmaslo_sm_nizkoe.Remont OR
  protections.Pmaslo_sm_vysokoe.Remont OR
  protections.Vibro_skorost_OPED_T1.Remont OR
  protections.Vibro_skorost_OPED_T2.Remont OR
  protections.Vibro_skorost_OYP_kolesa_ED_T3.Remont OR
  protections.Vibro_skorost_OP_kolesa_RH_T4.Remont OR
  protections.Vibro_skorost_OP_shesterni_RED_T5.Remont OR
  protections.Vibro_skorost_OP_shesterni_RED_T6.Remont OR
  protections.dPmaslo_gaz_less100.Remont OR
  protections.Reg_vozb_off.Remont OR
  protections.Fail_chastotnii_pusk.Remont OR
  protections.Off_avar_vikluchatel.Remont OR
  protections.AOKC_SHKC.Remont OR
  protections.AO_PRU.Remont OR
  protections.AO_ot_SHU.Remont OR
  protections.mvOff.Remont OR
  protections.Kran1_sdvig.Remont OR
  protections.Kran2_sdvig.Remont;
END_FUNCTION

FUNCTION ResetAllSignaling : BOOL
  VAR_IN_OUT
    protections : ProtectionsConfig;
  END_VAR

  IF protections.Topornogo_podshipnika_EDT_1.Signaling THEN
      resetAiProtection(protections.Topornogo_podshipnika_EDT_1);  END_IF;

  IF protections.Toy_podshipnika_EDT_2.Signaling THEN
      resetAiProtection(protections.Toy_podshipnika_EDT_2); END_IF;

  IF protections.Toy_podshipnika_kol_EDT_3.Signaling THEN
      resetAiProtection(protections.Toy_podshipnika_kol_EDT_3); END_IF;

  IF protections.Toy_podshipnika_kol_EDT_4.Signaling THEN
      resetAiProtection(protections.Toy_podshipnika_kol_EDT_4); END_IF;

  IF protections.To_podshipnika_shest_red_EDT_5.Signaling THEN
      resetAiProtection(protections.To_podshipnika_shest_red_EDT_5); END_IF;

  IF protections.To_podshipnika_shest_red_EDT_6.Signaling THEN
      resetAiProtection(protections.To_podshipnika_shest_red_EDT_6); END_IF;

  IF protections.To_podshipnika_N_EDT_7.Signaling THEN
      resetAiProtection(protections.To_podshipnika_N_EDT_7); END_IF;

  IF protections.To_podshipnika_svob_konca_EDT_8.Signaling THEN
      resetAiProtection(protections.To_podshipnika_svob_konca_EDT_8); END_IF;

  IF protections.Ty_podshipnika_rab_kol_EDT_9.Signaling THEN
      resetAiProtection(protections.Ty_podshipnika_rab_kol_EDT_9); END_IF;

  IF protections.Typornogo_podshipnika_nerab_kolodok_HT_10.Signaling THEN
      resetAiProtection(protections.Typornogo_podshipnika_nerab_kolodok_HT_10); END_IF;

  IF protections.Tgaza_na_vyhode_H.Signaling THEN
      resetAiProtection(protections.Tgaza_na_vyhode_H); END_IF;

  IF protections.Os_sdvig_nagnetatelja_plus.Signaling THEN
     resetAiProtection(protections.Os_sdvig_nagnetatelja_plus); END_IF;

  IF protections.Os_sdvig_nagnetatelja_minus.Signaling THEN
      resetAiProtection(protections.Os_sdvig_nagnetatelja_minus); END_IF;

  IF protections.Pgaza_na_vyhode_nagnetatelia_GPA_STOP.Signaling THEN
      resetAiProtection(protections.Pgaza_na_vyhode_nagnetatelia_GPA_STOP); END_IF;

  IF protections.Pgaza_na_vhode_nagnetatelia_GPA_STOP.Signaling THEN
      resetAiProtection(protections.Pgaza_na_vhode_nagnetatelia_GPA_STOP); END_IF;

  IF protections.Pgaza_na_vyhode_nagnetatelia.Signaling THEN
      resetAiProtection(protections.Pgaza_na_vyhode_nagnetatelia); END_IF;

  IF protections.dPmaslo_gaz.Signaling THEN
      resetAiProtection(protections.dPmaslo_gaz); END_IF;

  IF protections.Pmaslo_sm_nizkoe.Signaling THEN
      resetAiProtection(protections.Pmaslo_sm_nizkoe); END_IF;

  IF protections.Pmaslo_sm_vysokoe.Signaling THEN
      resetAiProtection(protections.Pmaslo_sm_vysokoe); END_IF;

  IF protections.Vibro_skorost_OPED_T1.Signaling THEN
      resetAiProtection(protections.Vibro_skorost_OPED_T1); END_IF;

  IF protections.Vibro_skorost_OPED_T2.Signaling THEN
      resetAiProtection(protections.Vibro_skorost_OPED_T2); END_IF;

  IF protections.Vibro_skorost_OYP_kolesa_ED_T3.Signaling THEN
      resetAiProtection(protections.Vibro_skorost_OYP_kolesa_ED_T3); END_IF;

  IF protections.Vibro_skorost_OP_kolesa_RH_T4.Signaling THEN
      resetAiProtection(protections.Vibro_skorost_OP_kolesa_RH_T4); END_IF;

  IF protections.Vibro_skorost_OP_shesterni_RED_T5.Signaling THEN
      resetAiProtection(protections.Vibro_skorost_OP_shesterni_RED_T5); END_IF;

  IF protections.Vibro_skorost_OP_shesterni_RED_T6.Signaling THEN
      resetAiProtection(protections.Vibro_skorost_OP_shesterni_RED_T6); END_IF;

  IF protections.dPmaslo_gaz_less100.Signaling THEN
      resetDiProtection(protections.dPmaslo_gaz_less100); END_IF;

  IF protections.Reg_vozb_off.Signaling THEN
      resetDiProtection(protections.Reg_vozb_off); END_IF;

  IF protections.Fail_chastotnii_pusk.Signaling THEN
      resetDiProtection(protections.Fail_chastotnii_pusk); END_IF;

  IF protections.Off_avar_vikluchatel.Signaling THEN
      resetDiProtection(protections.Off_avar_vikluchatel); END_IF;

  IF protections.AOKC_SHKC.Signaling THEN
      resetDiProtection(protections.AOKC_SHKC); END_IF;

  IF protections.AO_PRU.Signaling THEN
      resetDiProtection(protections.AO_PRU); END_IF;

  IF protections.AO_ot_SHU.Signaling THEN
      resetDiProtection(protections.AO_ot_SHU); END_IF;

  IF protections.mvOff.Signaling THEN
      resetDiProtection(protections.mvOff); END_IF;

  IF protections.Kran1_sdvig.Signaling THEN
      resetDiProtection(protections.Kran1_sdvig); END_IF;

  IF protections.Kran2_sdvig.Signaling THEN
      resetDiProtection(protections.Kran2_sdvig); END_IF;
END_FUNCTION

FUNCTION_BLOCK fb_ProtectionsManager
  VAR
    cmd : BYTE;
  END_VAR
  VAR_IN_OUT
    str_PM : struct_ProtectionsManager;
  END_VAR
  VAR
    lastCmd : BYTE;
    autoRunPriznak : BOOL;
    onInit : BOOL;
  END_VAR
  VAR_EXTERNAL
    protections : ProtectionsConfig;
  END_VAR
  VAR
    timerUnBlock : TON;
    timerAutoRun : TON;
    UnBlockPriznak : BOOL;
  END_VAR

  IF NOT onInit THEN

      autoRunProtections(protections);
  onInit:=TRUE;
  END_IF;

  str_PM.protectionInRemont:=anyProtectioninRemont(protections);

  cmd := str_PM.inCommand;

  IF cmd <> 0 AND lastCmd <> cmd then
                UnBlockPriznak:=TRUE;
  	CASE BYTE_TO_INT(cmd) OF

  		(*RestartAllSignaling*) 1: 	ResetAllSignaling(protections);
  				          autoRunPriznak:=TRUE;

  	        (*RestartAllProtections*) 2: 	ResetAllProtections(protections);
                                                    autoRunPriznak:=TRUE;

                        (*CheckProtections*)  3: 	RunAllProtections(protections);

  	         (*ResetAllProtections*)  4: 	ResetAllProtections(protections);

  	END_CASE;

  END_IF;
  lastCmd := cmd;
  timerUnBlock(IN:=UnBlockPriznak, PT:=T#1S);
  timerAutoRun(IN:=autoRunPriznak, PT:=T#500MS);

  IF timerAutoRun.Q THEN autoRunProtections(protections);
  END_IF;

  IF timerUnBlock.Q THEN
  lastCmd:= 0;
  str_PM.inCommand:=0;
  autoRunPriznak:=FALSE;
  UnBlockPriznak:=FALSE;
  END_IF;
END_FUNCTION_BLOCK

FUNCTION_BLOCK OPC_AI_INIT
  VAR_EXTERNAL
    AI_Tstali_statora_kanal_1_HL : LREAL;
    AI_Tstali_statora_kanal_1_LL : LREAL;
    AI_Tstali_statora_kanal_1_command : UINT;
    AI_Tstali_statora_kanal_1_newHL : LREAL;
    AI_Tstali_statora_kanal_1_newLL : LREAL;
    AI_Tstali_statora_kanal_1_status : UDINT;
    AI_Tstali_statora_kanal_1_value : LREAL;
    AI_Tstali_statora_kanal_1_HW : LREAL;
    AI_Tstali_statora_kanal_1_newHW : LREAL;
    AI_Tstali_statora_kanal_2_HL : LREAL;
    AI_Tstali_statora_kanal_2_LL : LREAL;
    AI_Tstali_statora_kanal_2_command : UINT;
    AI_Tstali_statora_kanal_2_newHL : LREAL;
    AI_Tstali_statora_kanal_2_newLL : LREAL;
    AI_Tstali_statora_kanal_2_status : UDINT;
    AI_Tstali_statora_kanal_2_value : LREAL;
    AI_Tstali_statora_kanal_2_HW : LREAL;
    AI_Tstali_statora_kanal_2_newHW : LREAL;
    AI_Tstali_statora_kanal_3_HL : LREAL;
    AI_Tstali_statora_kanal_3_LL : LREAL;
    AI_Tstali_statora_kanal_3_command : UINT;
    AI_Tstali_statora_kanal_3_newHL : LREAL;
    AI_Tstali_statora_kanal_3_newLL : LREAL;
    AI_Tstali_statora_kanal_3_status : UDINT;
    AI_Tstali_statora_kanal_3_value : LREAL;
    AI_Tstali_statora_kanal_3_HW : LREAL;
    AI_Tstali_statora_kanal_3_newHW : LREAL;
    AI_Tmedi_statora_kanal_1_HL : LREAL;
    AI_Tmedi_statora_kanal_1_LL : LREAL;
    AI_Tmedi_statora_kanal_1_command : UINT;
    AI_Tmedi_statora_kanal_1_newHL : LREAL;
    AI_Tmedi_statora_kanal_1_newLL : LREAL;
    AI_Tmedi_statora_kanal_1_status : UDINT;
    AI_Tmedi_statora_kanal_1_value : LREAL;
    AI_Tmedi_statora_kanal_1_HW : LREAL;
    AI_Tmedi_statora_kanal_1_newHW : LREAL;
    AI_Tmedi_statora_kanal_2_HL : LREAL;
    AI_Tmedi_statora_kanal_2_LL : LREAL;
    AI_Tmedi_statora_kanal_2_command : UINT;
    AI_Tmedi_statora_kanal_2_newHL : LREAL;
    AI_Tmedi_statora_kanal_2_newLL : LREAL;
    AI_Tmedi_statora_kanal_2_status : UDINT;
    AI_Tmedi_statora_kanal_2_value : LREAL;
    AI_Tmedi_statora_kanal_2_HW : LREAL;
    AI_Tmedi_statora_kanal_2_newHW : LREAL;
    AI_Tmedi_statora_kanal_3_HL : LREAL;
    AI_Tmedi_statora_kanal_3_LL : LREAL;
    AI_Tmedi_statora_kanal_3_command : UINT;
    AI_Tmedi_statora_kanal_3_newHL : LREAL;
    AI_Tmedi_statora_kanal_3_newLL : LREAL;
    AI_Tmedi_statora_kanal_3_status : UDINT;
    AI_Tmedi_statora_kanal_3_value : LREAL;
    AI_Tmedi_statora_kanal_3_HW : LREAL;
    AI_Tmedi_statora_kanal_3_newHW : LREAL;
    AI_Toporno_podshipnika_EDT_1_HL : LREAL;
    AI_Toporno_podshipnika_EDT_1_LL : LREAL;
    AI_Toporno_podshipnika_EDT_1_command : UINT;
    AI_Toporno_podshipnika_EDT_1_newHL : LREAL;
    AI_Toporno_podshipnika_EDT_1_newLL : LREAL;
    AI_Toporno_podshipnika_EDT_1_status : UDINT;
    AI_Toporno_podshipnika_EDT_1_value : LREAL;
    AI_Toporno_podshipnika_EDT_1_HW : LREAL;
    AI_Toporno_podshipnika_EDT_1_newHW : LREAL;
    AI_Toporno_podshipnika_EDT_1_HA : LREAL;
    AI_Toporno_podshipnika_EDT_1_newHA : LREAL;
    AI_Toy_podshipnika_EDT_2_HL : LREAL;
    AI_Toy_podshipnika_EDT_2_LL : LREAL;
    AI_Toy_podshipnika_EDT_2_command : UINT;
    AI_Toy_podshipnika_EDT_2_newHL : LREAL;
    AI_Toy_podshipnika_EDT_2_newLL : LREAL;
    AI_Toy_podshipnika_EDT_2_status : UDINT;
    AI_Toy_podshipnika_EDT_2_value : LREAL;
    AI_Toy_podshipnika_EDT_2_HW : LREAL;
    AI_Toy_podshipnika_EDT_2_newHW : LREAL;
    AI_Toy_podshipnika_EDT_2_HA : LREAL;
    AI_Toy_podshipnika_EDT_2_newHA : LREAL;
    AI_Toy_podshipnika_kol_EDT_3_HL : LREAL;
    AI_Toy_podshipnika_kol_EDT_3_LL : LREAL;
    AI_Toy_podshipnika_kol_EDT_3_command : UINT;
    AI_Toy_podshipnika_kol_EDT_3_newHL : LREAL;
    AI_Toy_podshipnika_kol_EDT_3_newLL : LREAL;
    AI_Toy_podshipnika_kol_EDT_3_status : UDINT;
    AI_Toy_podshipnika_kol_EDT_3_value : LREAL;
    AI_Toy_podshipnika_kol_EDT_3_HW : LREAL;
    AI_Toy_podshipnika_kol_EDT_3_newHW : LREAL;
    AI_Toy_podshipnika_kol_EDT_3_HA : LREAL;
    AI_Toy_podshipnika_kol_EDT_3_newHA : LREAL;
    AI_Toy_podshipnika_kol_EDT_4_HL : LREAL;
    AI_Toy_podshipnika_kol_EDT_4_LL : LREAL;
    AI_Toy_podshipnika_kol_EDT_4_command : UINT;
    AI_Toy_podshipnika_kol_EDT_4_newHL : LREAL;
    AI_Toy_podshipnika_kol_EDT_4_newLL : LREAL;
    AI_Toy_podshipnika_kol_EDT_4_status : UDINT;
    AI_Toy_podshipnika_kol_EDT_4_value : LREAL;
    AI_Toy_podshipnika_kol_EDT_4_HW : LREAL;
    AI_Toy_podshipnika_kol_EDT_4_newHW : LREAL;
    AI_Toy_podshipnika_kol_EDT_4_HA : LREAL;
    AI_Toy_podshipnika_kol_EDT_4_newHA : LREAL;
    AI_Toy_podshipnika_shest_red_EDT_5_HL : LREAL;
    AI_Toy_podshipnika_shest_red_EDT_5_LL : LREAL;
    AI_Toy_podshipnika_shest_red_EDT_5_command : UINT;
    AI_Toy_podshipnika_shest_red_EDT_5_newHL : LREAL;
    AI_Toy_podshipnika_shest_red_EDT_5_newLL : LREAL;
    AI_Toy_podshipnika_shest_red_EDT_5_status : UDINT;
    AI_Toy_podshipnika_shest_red_EDT_5_value : LREAL;
    AI_Toy_podshipnika_shest_red_EDT_5_HW : LREAL;
    AI_Toy_podshipnika_shest_red_EDT_5_newHW : LREAL;
    AI_Toy_podshipnika_shest_red_EDT_5_HA : LREAL;
    AI_Toy_podshipnika_shest_red_EDT_5_newHA : LREAL;
    AI_Ty_podshipnika_red_EDT_6_HL : LREAL;
    AI_Ty_podshipnika_red_EDT_6_LL : LREAL;
    AI_Ty_podshipnika_red_EDT_6_command : UINT;
    AI_Ty_podshipnika_red_EDT_6_newHL : LREAL;
    AI_Ty_podshipnika_red_EDT_6_newLL : LREAL;
    AI_Ty_podshipnika_red_EDT_6_status : UDINT;
    AI_Ty_podshipnika_red_EDT_6_value : LREAL;
    AI_Ty_podshipnika_red_EDT_6_HW : LREAL;
    AI_Ty_podshipnika_red_EDT_6_newHW : LREAL;
    AI_Ty_podshipnika_red_EDT_6_HA : LREAL;
    AI_Ty_podshipnika_red_EDT_6_newHA : LREAL;
    AI_Ty_podshipnika_nagnet_EDT_7_1_HL : LREAL;
    AI_Ty_podshipnika_nagnet_EDT_7_1_LL : LREAL;
    AI_Ty_podshipnika_nagnet_EDT_7_1_command : UINT;
    AI_Ty_podshipnika_nagnet_EDT_7_1_newHL : LREAL;
    AI_Ty_podshipnika_nagnet_EDT_7_1_newLL : LREAL;
    AI_Ty_podshipnika_nagnet_EDT_7_1_status : UDINT;
    AI_Ty_podshipnika_nagnet_EDT_7_1_value : LREAL;
    AI_Ty_podshipnika_nagnet_EDT_7_1_HW : LREAL;
    AI_Ty_podshipnika_nagnet_EDT_7_1_newHW : LREAL;
    AI_Ty_podshipnika_nagnet_EDT_7_1_HA : LREAL;
    AI_Ty_podshipnika_nagnet_EDT_7_1_newHA : LREAL;
    AI_Ty_podshipnika_nagnet_EDT_7_2_HL : LREAL;
    AI_Ty_podshipnika_nagnet_EDT_7_2_LL : LREAL;
    AI_Ty_podshipnika_nagnet_EDT_7_2_command : UINT;
    AI_Ty_podshipnika_nagnet_EDT_7_2_newHL : LREAL;
    AI_Ty_podshipnika_nagnet_EDT_7_2_newLL : LREAL;
    AI_Ty_podshipnika_nagnet_EDT_7_2_status : UDINT;
    AI_Ty_podshipnika_nagnet_EDT_7_2_value : LREAL;
    AI_Ty_podshipnika_nagnet_EDT_7_2_HW : LREAL;
    AI_Ty_podshipnika_nagnet_EDT_7_2_newHW : LREAL;
    AI_Ty_podshipnika_nagnet_EDT_7_2_HA : LREAL;
    AI_Ty_podshipnika_nagnet_EDT_7_2_newHA : LREAL;
    AI_Toy_podshipnika_svobod_konca_EDT_8_1_HL : LREAL;
    AI_Toy_podshipnika_svobod_konca_EDT_8_1_LL : LREAL;
    AI_Toy_podshipnika_svobod_konca_EDT_8_1_command : UINT;
    AI_Toy_podshipnika_svobod_konca_EDT_8_1_newHL : LREAL;
    AI_Toy_podshipnika_svobod_konca_EDT_8_1_newLL : LREAL;
    AI_Toy_podshipnika_svobod_konca_EDT_8_1_status : UDINT;
    AI_Toy_podshipnika_svobod_konca_EDT_8_1_value : LREAL;
    AI_Toy_podshipnika_svobod_konca_EDT_8_1_HW : LREAL;
    AI_Toy_podshipnika_svobod_konca_EDT_8_1_newHW : LREAL;
    AI_Toy_podshipnika_svobod_konca_EDT_8_1_HA : LREAL;
    AI_Toy_podshipnika_svobod_konca_EDT_8_1_newHA : LREAL;
    AI_Toy_podshipnika_svobod_konca_EDT_8_2_HL : LREAL;
    AI_Toy_podshipnika_svobod_konca_EDT_8_2_LL : LREAL;
    AI_Toy_podshipnika_svobod_konca_EDT_8_2_command : UINT;
    AI_Toy_podshipnika_svobod_konca_EDT_8_2_newHL : LREAL;
    AI_Toy_podshipnika_svobod_konca_EDT_8_2_newLL : LREAL;
    AI_Toy_podshipnika_svobod_konca_EDT_8_2_status : UDINT;
    AI_Toy_podshipnika_svobod_konca_EDT_8_2_value : LREAL;
    AI_Toy_podshipnika_svobod_konca_EDT_8_2_HW : LREAL;
    AI_Toy_podshipnika_svobod_konca_EDT_8_2_newHW : LREAL;
    AI_Toy_podshipnika_svobod_konca_EDT_8_2_HA : LREAL;
    AI_Toy_podshipnika_svobod_konca_EDT_8_2_newHA : LREAL;
    AI_Toy_podshipnika_rab_kol_EDT_9_1_HL : LREAL;
    AI_Toy_podshipnika_rab_kol_EDT_9_1_LL : LREAL;
    AI_Toy_podshipnika_rab_kol_EDT_9_1_command : UINT;
    AI_Toy_podshipnika_rab_kol_EDT_9_1_newHL : LREAL;
    AI_Toy_podshipnika_rab_kol_EDT_9_1_newLL : LREAL;
    AI_Toy_podshipnika_rab_kol_EDT_9_1_status : UDINT;
    AI_Toy_podshipnika_rab_kol_EDT_9_1_value : LREAL;
    AI_Toy_podshipnika_rab_kol_EDT_9_1_HW : LREAL;
    AI_Toy_podshipnika_rab_kol_EDT_9_1_newHW : LREAL;
    AI_Toy_podshipnika_rab_kol_EDT_9_1_HA : LREAL;
    AI_Toy_podshipnika_rab_kol_EDT_9_1_newHA : LREAL;
    AI_Toy_podshipnika_rab_kol_EDT_9_2_HL : LREAL;
    AI_Toy_podshipnika_rab_kol_EDT_9_2_LL : LREAL;
    AI_Toy_podshipnika_rab_kol_EDT_9_2_command : UINT;
    AI_Toy_podshipnika_rab_kol_EDT_9_2_newHL : LREAL;
    AI_Toy_podshipnika_rab_kol_EDT_9_2_newLL : LREAL;
    AI_Toy_podshipnika_rab_kol_EDT_9_2_status : UDINT;
    AI_Toy_podshipnika_rab_kol_EDT_9_2_value : LREAL;
    AI_Toy_podshipnika_rab_kol_EDT_9_2_HW : LREAL;
    AI_Toy_podshipnika_rab_kol_EDT_9_2_newHW : LREAL;
    AI_Toy_podshipnika_rab_kol_EDT_9_2_HA : LREAL;
    AI_Toy_podshipnika_rab_kol_EDT_9_2_newHA : LREAL;
    AI_Toy_podshipnika_nerab_kol_EDT_10_1_HL : LREAL;
    AI_Toy_podshipnika_nerab_kol_EDT_10_1_LL : LREAL;
    AI_Toy_podshipnika_nerab_kol_EDT_10_1_command : UINT;
    AI_Toy_podshipnika_nerab_kol_EDT_10_1_newHL : LREAL;
    AI_Toy_podshipnika_nerab_kol_EDT_10_1_newLL : LREAL;
    AI_Toy_podshipnika_nerab_kol_EDT_10_1_status : UDINT;
    AI_Toy_podshipnika_nerab_kol_EDT_10_1_value : LREAL;
    AI_Toy_podshipnika_nerab_kol_EDT_10_1_HW : LREAL;
    AI_Toy_podshipnika_nerab_kol_EDT_10_1_newHW : LREAL;
    AI_Toy_podshipnika_nerab_kol_EDT_10_1_HA : LREAL;
    AI_Toy_podshipnika_nerab_kol_EDT_10_1_newHA : LREAL;
    AI_Toy_podshipnika_nerab_kol_EDT_10_2_HL : LREAL;
    AI_Toy_podshipnika_nerab_kol_EDT_10_2_LL : LREAL;
    AI_Toy_podshipnika_nerab_kol_EDT_10_2_command : UINT;
    AI_Toy_podshipnika_nerab_kol_EDT_10_2_newHL : LREAL;
    AI_Toy_podshipnika_nerab_kol_EDT_10_2_newLL : LREAL;
    AI_Toy_podshipnika_nerab_kol_EDT_10_2_status : UDINT;
    AI_Toy_podshipnika_nerab_kol_EDT_10_2_value : LREAL;
    AI_Toy_podshipnika_nerab_kol_EDT_10_2_HW : LREAL;
    AI_Toy_podshipnika_nerab_kol_EDT_10_2_newHW : LREAL;
    AI_Toy_podshipnika_nerab_kol_EDT_10_2_HA : LREAL;
    AI_Toy_podshipnika_nerab_kol_EDT_10_2_newHA : LREAL;
    AI_Tholodnogo_vozduha_ED_kanal_1_HL : LREAL;
    AI_Tholodnogo_vozduha_ED_kanal_1_LL : LREAL;
    AI_Tholodnogo_vozduha_ED_kanal_1_command : UINT;
    AI_Tholodnogo_vozduha_ED_kanal_1_newHL : LREAL;
    AI_Tholodnogo_vozduha_ED_kanal_1_newLL : LREAL;
    AI_Tholodnogo_vozduha_ED_kanal_1_status : UDINT;
    AI_Tholodnogo_vozduha_ED_kanal_1_value : LREAL;
    AI_Tholodnogo_vozduha_ED_kanal_1_HW : LREAL;
    AI_Tholodnogo_vozduha_ED_kanal_1_newHW : LREAL;
    AI_Tholodnogo_vozduha_ED_kanal_2_HL : LREAL;
    AI_Tholodnogo_vozduha_ED_kanal_2_LL : LREAL;
    AI_Tholodnogo_vozduha_ED_kanal_2_command : UINT;
    AI_Tholodnogo_vozduha_ED_kanal_2_newHL : LREAL;
    AI_Tholodnogo_vozduha_ED_kanal_2_newLL : LREAL;
    AI_Tholodnogo_vozduha_ED_kanal_2_status : UDINT;
    AI_Tholodnogo_vozduha_ED_kanal_2_value : LREAL;
    AI_Tholodnogo_vozduha_ED_kanal_2_HW : LREAL;
    AI_Tholodnogo_vozduha_ED_kanal_2_newHW : LREAL;
    AI_Tgorjachego_vozduha_ED_kanal_1_HL : LREAL;
    AI_Tgorjachego_vozduha_ED_kanal_1_LL : LREAL;
    AI_Tgorjachego_vozduha_ED_kanal_1_command : UINT;
    AI_Tgorjachego_vozduha_ED_kanal_1_newHL : LREAL;
    AI_Tgorjachego_vozduha_ED_kanal_1_newLL : LREAL;
    AI_Tgorjachego_vozduha_ED_kanal_1_status : UDINT;
    AI_Tgorjachego_vozduha_ED_kanal_1_value : LREAL;
    AI_Tgorjachego_vozduha_ED_kanal_1_HW : LREAL;
    AI_Tgorjachego_vozduha_ED_kanal_1_newHW : LREAL;
    AI_Tgorjachego_vozduha_ED_kanal_2_HL : LREAL;
    AI_Tgorjachego_vozduha_ED_kanal_2_LL : LREAL;
    AI_Tgorjachego_vozduha_ED_kanal_2_command : UINT;
    AI_Tgorjachego_vozduha_ED_kanal_2_newHL : LREAL;
    AI_Tgorjachego_vozduha_ED_kanal_2_newLL : LREAL;
    AI_Tgorjachego_vozduha_ED_kanal_2_status : UDINT;
    AI_Tgorjachego_vozduha_ED_kanal_2_value : LREAL;
    AI_Tgorjachego_vozduha_ED_kanal_2_HW : LREAL;
    AI_Tgorjachego_vozduha_ED_kanal_2_newHW : LREAL;
    AI_Tnarujnogo_vozduha_HL : LREAL;
    AI_Tnarujnogo_vozduha_LL : LREAL;
    AI_Tnarujnogo_vozduha_command : UINT;
    AI_Tnarujnogo_vozduha_newHL : LREAL;
    AI_Tnarujnogo_vozduha_newLL : LREAL;
    AI_Tnarujnogo_vozduha_status : UDINT;
    AI_Tnarujnogo_vozduha_value : LREAL;
    AI_Tnarujnogo_vozduha_HW : LREAL;
    AI_Tnarujnogo_vozduha_newHW : LREAL;
    AI_Tgaza_na_vhode_H_HL : LREAL;
    AI_Tgaza_na_vhode_H_LL : LREAL;
    AI_Tgaza_na_vhode_H_command : UINT;
    AI_Tgaza_na_vhode_H_newHL : LREAL;
    AI_Tgaza_na_vhode_H_newLL : LREAL;
    AI_Tgaza_na_vhode_H_status : UDINT;
    AI_Tgaza_na_vhode_H_value : LREAL;
    AI_Tgaza_na_vhode_H_HW : LREAL;
    AI_Tgaza_na_vhode_H_newHW : LREAL;
    AI_Tgaza_na_vyhode_H_HL : LREAL;
    AI_Tgaza_na_vyhode_H_LL : LREAL;
    AI_Tgaza_na_vyhode_H_command : UINT;
    AI_Tgaza_na_vyhode_H_newHL : LREAL;
    AI_Tgaza_na_vyhode_H_newLL : LREAL;
    AI_Tgaza_na_vyhode_H_status : UDINT;
    AI_Tgaza_na_vyhode_H_value : LREAL;
    AI_Tgaza_na_vyhode_H_HW : LREAL;
    AI_Tgaza_na_vyhode_H_newHW : LREAL;
    AI_Tgaza_na_vyhode_H_HA : LREAL;
    AI_Tgaza_na_vyhode_H_newHA : LREAL;
    AI_Tmasla_do_AVOM_HL : LREAL;
    AI_Tmasla_do_AVOM_LL : LREAL;
    AI_Tmasla_do_AVOM_command : UINT;
    AI_Tmasla_do_AVOM_newHL : LREAL;
    AI_Tmasla_do_AVOM_newLL : LREAL;
    AI_Tmasla_do_AVOM_status : UDINT;
    AI_Tmasla_do_AVOM_value : LREAL;
    AI_Tmasla_do_AVOM_HW : LREAL;
    AI_Tmasla_do_AVOM_newHW : LREAL;
    AI_Tmasla_posle_AVOM_HL : LREAL;
    AI_Tmasla_posle_AVOM_LL : LREAL;
    AI_Tmasla_posle_AVOM_command : UINT;
    AI_Tmasla_posle_AVOM_newHL : LREAL;
    AI_Tmasla_posle_AVOM_newLL : LREAL;
    AI_Tmasla_posle_AVOM_status : UDINT;
    AI_Tmasla_posle_AVOM_value : LREAL;
    AI_Tmasla_posle_AVOM_HW : LREAL;
    AI_Tmasla_posle_AVOM_newHW : LREAL;
    AI_Tmasla_MB_HL : LREAL;
    AI_Tmasla_MB_LL : LREAL;
    AI_Tmasla_MB_command : UINT;
    AI_Tmasla_MB_newHL : LREAL;
    AI_Tmasla_MB_newLL : LREAL;
    AI_Tmasla_MB_status : UDINT;
    AI_Tmasla_MB_value : LREAL;
    AI_Tmasla_MB_LW : LREAL;
    AI_Tmasla_MB_newLW : LREAL;
    AI_Tmasla_MB_TEN_HL : LREAL;
    AI_Tmasla_MB_TEN_LL : LREAL;
    AI_Tmasla_MB_TEN_command : UINT;
    AI_Tmasla_MB_TEN_newHL : LREAL;
    AI_Tmasla_MB_TEN_newLL : LREAL;
    AI_Tmasla_MB_TEN_status : UDINT;
    AI_Tmasla_MB_TEN_value : LREAL;
    AI_Tmasla_MB_TEN_HW : LREAL;
    AI_Tmasla_MB_TEN_newHW : LREAL;
    AI_Tshu_HL : LREAL;
    AI_Tshu_LL : LREAL;
    AI_Tshu_command : UINT;
    AI_Tshu_newHL : LREAL;
    AI_Tshu_newLL : LREAL;
    AI_Tshu_status : UDINT;
    AI_Tshu_value : LREAL;
    AI_Pmaslo_sm_nizkoe_HL : LREAL;
    AI_Pmaslo_sm_nizkoe_LL : LREAL;
    AI_Pmaslo_sm_nizkoe_command : UINT;
    AI_Pmaslo_sm_nizkoe_newHL : LREAL;
    AI_Pmaslo_sm_nizkoe_newLL : LREAL;
    AI_Pmaslo_sm_nizkoe_status : UDINT;
    AI_Pmaslo_sm_nizkoe_value : LREAL;
    AI_Pmaslo_sm_nizkoe_LW : LREAL;
    AI_Pmaslo_sm_nizkoe_newLW : LREAL;
    AI_Pmaslo_sm_nizkoe_LA : LREAL;
    AI_Pmaslo_sm_nizkoe_newLA : LREAL;
    AI_Pmaslo_sm_vysokoe_HL : LREAL;
    AI_Pmaslo_sm_vysokoe_LL : LREAL;
    AI_Pmaslo_sm_vysokoe_command : UINT;
    AI_Pmaslo_sm_vysokoe_newHL : LREAL;
    AI_Pmaslo_sm_vysokoe_newLL : LREAL;
    AI_Pmaslo_sm_vysokoe_status : UDINT;
    AI_Pmaslo_sm_vysokoe_value : LREAL;
    AI_Pmaslo_sm_vysokoe_LW : LREAL;
    AI_Pmaslo_sm_vysokoe_newLW : LREAL;
    AI_Pmaslo_sm_vysokoe_LA : LREAL;
    AI_Pmaslo_sm_vysokoe_newLA : LREAL;
    AI_Pmasla_posle_GNS_HL : LREAL;
    AI_Pmasla_posle_GNS_LL : LREAL;
    AI_Pmasla_posle_GNS_command : UINT;
    AI_Pmasla_posle_GNS_newHL : LREAL;
    AI_Pmasla_posle_GNS_newLL : LREAL;
    AI_Pmasla_posle_GNS_status : UDINT;
    AI_Pmasla_posle_GNS_value : LREAL;
    AI_Pmasla_posle_GNS_HW : LREAL;
    AI_Pmasla_posle_GNS_newHW : LREAL;
    AI_Pmasla_posle_GNS_LW : LREAL;
    AI_Pmasla_posle_GNS_newLW : LREAL;
    AI_Pmasla_posle_NU_HL : LREAL;
    AI_Pmasla_posle_NU_LL : LREAL;
    AI_Pmasla_posle_NU_command : UINT;
    AI_Pmasla_posle_NU_newHL : LREAL;
    AI_Pmasla_posle_NU_newLL : LREAL;
    AI_Pmasla_posle_NU_status : UDINT;
    AI_Pmasla_posle_NU_value : LREAL;
    AI_Pmasla_posle_NU_LW : LREAL;
    AI_Pmasla_posle_NU_newLW : LREAL;
    AI_Pgaza_na_vhode_nagnetatelia_HL : LREAL;
    AI_Pgaza_na_vhode_nagnetatelia_LL : LREAL;
    AI_Pgaza_na_vhode_nagnetatelia_command : UINT;
    AI_Pgaza_na_vhode_nagnetatelia_newHL : LREAL;
    AI_Pgaza_na_vhode_nagnetatelia_newLL : LREAL;
    AI_Pgaza_na_vhode_nagnetatelia_status : UDINT;
    AI_Pgaza_na_vhode_nagnetatelia_value : LREAL;
    AI_Pgaza_na_vhode_nagnetatelia_LW : LREAL;
    AI_Pgaza_na_vhode_nagnetatelia_newLW : LREAL;
    AI_Pgaza_na_vyhode_nagnetatelia_HL : LREAL;
    AI_Pgaza_na_vyhode_nagnetatelia_LL : LREAL;
    AI_Pgaza_na_vyhode_nagnetatelia_command : UINT;
    AI_Pgaza_na_vyhode_nagnetatelia_newHL : LREAL;
    AI_Pgaza_na_vyhode_nagnetatelia_newLL : LREAL;
    AI_Pgaza_na_vyhode_nagnetatelia_status : UDINT;
    AI_Pgaza_na_vyhode_nagnetatelia_value : LREAL;
    AI_Pgaza_na_vyhode_nagnetatelia_HW : LREAL;
    AI_Pgaza_na_vyhode_nagnetatelia_newHW : LREAL;
    AI_Pgaza_na_vyhode_nagnetatelia_HA : LREAL;
    AI_Pgaza_na_vyhode_nagnetatelia_newHA : LREAL;
    AI_Pimpuls_gaz_HL : LREAL;
    AI_Pimpuls_gaz_LL : LREAL;
    AI_Pimpuls_gaz_command : UINT;
    AI_Pimpuls_gaz_newHL : LREAL;
    AI_Pimpuls_gaz_newLL : LREAL;
    AI_Pimpuls_gaz_status : UDINT;
    AI_Pimpuls_gaz_value : LREAL;
    AI_Pimpuls_gaz_LW : LREAL;
    AI_Pimpuls_gaz_newLW : LREAL;
    AI_dPgaza_na_maslo_filtre_HL : LREAL;
    AI_dPgaza_na_maslo_filtre_LL : LREAL;
    AI_dPgaza_na_maslo_filtre_command : UINT;
    AI_dPgaza_na_maslo_filtre_newHL : LREAL;
    AI_dPgaza_na_maslo_filtre_newLL : LREAL;
    AI_dPgaza_na_maslo_filtre_status : UDINT;
    AI_dPgaza_na_maslo_filtre_value : LREAL;
    AI_dPgaza_na_maslo_filtre_HW : LREAL;
    AI_dPgaza_na_maslo_filtre_newHW : LREAL;
    AI_dPgaza_na_konfuzore_HL : LREAL;
    AI_dPgaza_na_konfuzore_LL : LREAL;
    AI_dPgaza_na_konfuzore_command : UINT;
    AI_dPgaza_na_konfuzore_newHL : LREAL;
    AI_dPgaza_na_konfuzore_newLL : LREAL;
    AI_dPgaza_na_konfuzore_status : UDINT;
    AI_dPgaza_na_konfuzore_value : LREAL;
    AI_dPgaza_na_konfuzore_LW : LREAL;
    AI_dPgaza_na_konfuzore_newLW : LREAL;
    AI_dPmaslo_gaz_HL : LREAL;
    AI_dPmaslo_gaz_LL : LREAL;
    AI_dPmaslo_gaz_command : UINT;
    AI_dPmaslo_gaz_newHL : LREAL;
    AI_dPmaslo_gaz_newLL : LREAL;
    AI_dPmaslo_gaz_status : UDINT;
    AI_dPmaslo_gaz_value : LREAL;
    AI_dPmaslo_gaz_LW : LREAL;
    AI_dPmaslo_gaz_newLW : LREAL;
    AI_dPmaslo_gaz_LA : LREAL;
    AI_dPmaslo_gaz_newLA : LREAL;
    AI_Os_sdvig_nagnetatelja_plus_HL : LREAL;
    AI_Os_sdvig_nagnetatelja_plus_LL : LREAL;
    AI_Os_sdvig_nagnetatelja_plus_command : UINT;
    AI_Os_sdvig_nagnetatelja_plus_newHL : LREAL;
    AI_Os_sdvig_nagnetatelja_plus_newLL : LREAL;
    AI_Os_sdvig_nagnetatelja_plus_status : UDINT;
    AI_Os_sdvig_nagnetatelja_plus_value : LREAL;
    AI_Os_sdvig_nagnetatelja_plus_HW : LREAL;
    AI_Os_sdvig_nagnetatelja_plus_newHW : LREAL;
    AI_Os_sdvig_nagnetatelja_plus_HA : LREAL;
    AI_Os_sdvig_nagnetatelja_plus_newHA : LREAL;
    AI_Os_sdvig_nagnetatelja_minus_HL : LREAL;
    AI_Os_sdvig_nagnetatelja_minus_LL : LREAL;
    AI_Os_sdvig_nagnetatelja_minus_command : UINT;
    AI_Os_sdvig_nagnetatelja_minus_newHL : LREAL;
    AI_Os_sdvig_nagnetatelja_minus_newLL : LREAL;
    AI_Os_sdvig_nagnetatelja_minus_status : UDINT;
    AI_Os_sdvig_nagnetatelja_minus_value : LREAL;
    AI_Os_sdvig_nagnetatelja_minus_LW : LREAL;
    AI_Os_sdvig_nagnetatelja_minus_newLW : LREAL;
    AI_Os_sdvig_nagnetatelja_minus_LA : LREAL;
    AI_Os_sdvig_nagnetatelja_minus_newLA : LREAL;
    AI_Yroven_masla_MB_HL : LREAL;
    AI_Yroven_masla_MB_LL : LREAL;
    AI_Yroven_masla_MB_command : UINT;
    AI_Yroven_masla_MB_newHL : LREAL;
    AI_Yroven_masla_MB_newLL : LREAL;
    AI_Yroven_masla_MB_status : UDINT;
    AI_Yroven_masla_MB_value : LREAL;
    AI_Yroven_masla_MB_LW : LREAL;
    AI_Yroven_masla_MB_newLW : LREAL;
    AI_Kontrol_per_220V_HL : LREAL;
    AI_Kontrol_per_220V_LL : LREAL;
    AI_Kontrol_per_220V_command : UINT;
    AI_Kontrol_per_220V_newHL : LREAL;
    AI_Kontrol_per_220V_newLL : LREAL;
    AI_Kontrol_per_220V_status : UDINT;
    AI_Kontrol_per_220V_value : LREAL;
    AI_Kontrol_per_220V_HW : LREAL;
    AI_Kontrol_per_220V_newHW : LREAL;
    AI_Kontrol_per_220V_LW : LREAL;
    AI_Kontrol_per_220V_newLW : LREAL;
    AI_Kontrol_post_220V_HL : LREAL;
    AI_Kontrol_post_220V_LL : LREAL;
    AI_Kontrol_post_220V_command : UINT;
    AI_Kontrol_post_220V_newHL : LREAL;
    AI_Kontrol_post_220V_newLL : LREAL;
    AI_Kontrol_post_220V_status : UDINT;
    AI_Kontrol_post_220V_value : LREAL;
    AI_Kontrol_post_220V_HW : LREAL;
    AI_Kontrol_post_220V_newHW : LREAL;
    AI_Kontrol_post_220V_LW : LREAL;
    AI_Kontrol_post_220V_newLW : LREAL;
    AI_Tok_statora_HL : LREAL;
    AI_Tok_statora_LL : LREAL;
    AI_Tok_statora_command : UINT;
    AI_Tok_statora_newHL : LREAL;
    AI_Tok_statora_newLL : LREAL;
    AI_Tok_statora_status : UDINT;
    AI_Tok_statora_value : LREAL;
    AI_Tok_statora_LW : LREAL;
    AI_Tok_statora_newLW : LREAL;
    AI_Vibro_skorost_OPED_T1_HL : LREAL;
    AI_Vibro_skorost_OPED_T1_LL : LREAL;
    AI_Vibro_skorost_OPED_T1_command : UINT;
    AI_Vibro_skorost_OPED_T1_newHL : LREAL;
    AI_Vibro_skorost_OPED_T1_newLL : LREAL;
    AI_Vibro_skorost_OPED_T1_status : UDINT;
    AI_Vibro_skorost_OPED_T1_value : LREAL;
    AI_Vibro_skorost_OPED_T1_HW : LREAL;
    AI_Vibro_skorost_OPED_T1_newHW : LREAL;
    AI_Vibro_skorost_OPED_T1_HA : LREAL;
    AI_Vibro_skorost_OPED_T1_newHA : LREAL;
    AI_Vibro_skorost_OYPED_T2_HL : LREAL;
    AI_Vibro_skorost_OYPED_T2_LL : LREAL;
    AI_Vibro_skorost_OYPED_T2_command : UINT;
    AI_Vibro_skorost_OYPED_T2_newHL : LREAL;
    AI_Vibro_skorost_OYPED_T2_newLL : LREAL;
    AI_Vibro_skorost_OYPED_T2_status : UDINT;
    AI_Vibro_skorost_OYPED_T2_value : LREAL;
    AI_Vibro_skorost_OYPED_T2_HW : LREAL;
    AI_Vibro_skorost_OYPED_T2_newHW : LREAL;
    AI_Vibro_skorost_OYPED_T2_HA : LREAL;
    AI_Vibro_skorost_OYPED_T2_newHA : LREAL;
    AI_Vibro_skorost_OYP_kolesa_ED_T3_HL : LREAL;
    AI_Vibro_skorost_OYP_kolesa_ED_T3_LL : LREAL;
    AI_Vibro_skorost_OYP_kolesa_ED_T3_command : UINT;
    AI_Vibro_skorost_OYP_kolesa_ED_T3_newHL : LREAL;
    AI_Vibro_skorost_OYP_kolesa_ED_T3_newLL : LREAL;
    AI_Vibro_skorost_OYP_kolesa_ED_T3_status : UDINT;
    AI_Vibro_skorost_OYP_kolesa_ED_T3_value : LREAL;
    AI_Vibro_skorost_OYP_kolesa_ED_T3_HW : LREAL;
    AI_Vibro_skorost_OYP_kolesa_ED_T3_newHW : LREAL;
    AI_Vibro_skorost_OYP_kolesa_ED_T3_HA : LREAL;
    AI_Vibro_skorost_OYP_kolesa_ED_T3_newHA : LREAL;
    AI_Vibro_skorost_OP_kolesa_RH_T4_HL : LREAL;
    AI_Vibro_skorost_OP_kolesa_RH_T4_LL : LREAL;
    AI_Vibro_skorost_OP_kolesa_RH_T4_command : UINT;
    AI_Vibro_skorost_OP_kolesa_RH_T4_newHL : LREAL;
    AI_Vibro_skorost_OP_kolesa_RH_T4_newLL : LREAL;
    AI_Vibro_skorost_OP_kolesa_RH_T4_status : UDINT;
    AI_Vibro_skorost_OP_kolesa_RH_T4_value : LREAL;
    AI_Vibro_skorost_OP_kolesa_RH_T4_HW : LREAL;
    AI_Vibro_skorost_OP_kolesa_RH_T4_newHW : LREAL;
    AI_Vibro_skorost_OP_kolesa_RH_T4_HA : LREAL;
    AI_Vibro_skorost_OP_kolesa_RH_T4_newHA : LREAL;
    AI_Vibro_skorost_OP_shesterni_RED_T5_HL : LREAL;
    AI_Vibro_skorost_OP_shesterni_RED_T5_LL : LREAL;
    AI_Vibro_skorost_OP_shesterni_RED_T5_command : UINT;
    AI_Vibro_skorost_OP_shesterni_RED_T5_newHL : LREAL;
    AI_Vibro_skorost_OP_shesterni_RED_T5_newLL : LREAL;
    AI_Vibro_skorost_OP_shesterni_RED_T5_status : UDINT;
    AI_Vibro_skorost_OP_shesterni_RED_T5_value : LREAL;
    AI_Vibro_skorost_OP_shesterni_RED_T5_HW : LREAL;
    AI_Vibro_skorost_OP_shesterni_RED_T5_newHW : LREAL;
    AI_Vibro_skorost_OP_shesterni_RED_T5_HA : LREAL;
    AI_Vibro_skorost_OP_shesterni_RED_T5_newHA : LREAL;
    AI_Vibro_skorost_OP_shesterni_RED_T6_HL : LREAL;
    AI_Vibro_skorost_OP_shesterni_RED_T6_LL : LREAL;
    AI_Vibro_skorost_OP_shesterni_RED_T6_command : UINT;
    AI_Vibro_skorost_OP_shesterni_RED_T6_newHL : LREAL;
    AI_Vibro_skorost_OP_shesterni_RED_T6_newLL : LREAL;
    AI_Vibro_skorost_OP_shesterni_RED_T6_status : UDINT;
    AI_Vibro_skorost_OP_shesterni_RED_T6_value : LREAL;
    AI_Vibro_skorost_OP_shesterni_RED_T6_HW : LREAL;
    AI_Vibro_skorost_OP_shesterni_RED_T6_newHW : LREAL;
    AI_Vibro_skorost_OP_shesterni_RED_T6_HA : LREAL;
    AI_Vibro_skorost_OP_shesterni_RED_T6_newHA : LREAL;
  END_VAR
